// ---- POUs/FBs/FanucKardex/DUTs/ST_Kardex_Robot_Control.TcDUT
TYPE ST_Kardex_Robot_Control :
STRUCT
(*-----=== Byte 01 ===-----*)
	bImmediateStop			:BIT;				// 01.1	Immediate stop
	bHold					:BIT;				// 01.2	Temporary stop
	bSafeSpeed				:BIT;				// 01.3	Safe speed
	bCycleStop				:BIT;				// 01.4	Cycle stop
	bReset					:BIT;				// 01.5	External reset
	bStart					:BIT;				// 01.6	Start
	bHome					:BIT;				// 01.7	Return to home position
	bEnable					:BIT;				// 01.8	Operation enable

(*-----=== Byte 02 ===-----*)
//	nProgNumberSelection	:BYTE;
	bPNS1					:BIT;				// 02.1	Program  number selection
	bPNS2					:BIT;				// 02.2	Program  number selection
	bPNS3					:BIT;				// 02.3	Program  number selection
	bPNS4					:BIT;				// 02.4	Program  number selection
	bPNS5					:BIT;				// 02.5	Program  number selection
	bPNS6					:BIT;				// 02.6	Program  number selection
	bPNS7					:BIT;				// 02.7	Program  number selection
	bPNS8					:BIT;				// 02.8	Program  number selection

(*-----=== Byte 03 ===-----*)
	bPnsStrobe				:BIT;				// 03.1	PNS strobe
	bProdStart				:BIT;				// 03.2	Start of automatic operation
	bZoneEnable				:BIT;				// 03.3	Ez mindig jön kivéve ha vész van
	bServiceEnd				:BIT;				// 03.4	Szervíz üzemmód vége
	{attribute 'hide'}
	_reserved_03_05			:BIT;
	{attribute 'hide'}
	_reserved_03_06			:BIT;
	{attribute 'hide'}
	_reserved_03_07			:BIT;		
	{attribute 'hide'}
	_reserved_03_08			:BIT;		
	
(*-----=== Byte 04 ===-----*)
	{attribute 'hide'}
	_reserved_04			:BYTE;				

(*-----=== Byte 05 ===-----*)
	bKardex_Reset			:BIT;				// 05.1	Robot kardex-be mehet RESET
	bHolder_Reset			:BIT;				// 05.2	Robot Mir-1-be mehet RESET
	bMir_Reset				:BIT;				// 05.3	Robot Mir-2-be mehet RESET
	bPuffer_Reset			:BIT;				// 05.4	Robot pufferbe mehet RESET
	bStrip_1_Reset			:BIT;				// 05.5	Robot szalag-1-be mehet RESET
	bStrip_2_Reset			:BIT;				// 05.6	Robot szalag-2-be mehet RESET
	bStrip_3_Reset			:BIT;				// 05.7	Robot szalag-3-be mehet RESET	
	{attribute 'hide'}
	_reserved_05_08			:BIT;
	
(*-----=== Byte 06 ===-----*)
	{attribute 'hide'}
	_reserved_06			:BYTE;				
	
(*-----=== Byte 07 ===-----*)
	bNotCorrectPrg_Reset			:BIT;				// 07.1	Nem megfelelő mozgási program RESET
	bNotProductOnRobot_Reset		:BIT;				// 07.2	Mozgási program nem hajtható végre, mert a robotnál nincs termék RESET
	bProductOnRobot_Reset			:BIT;				// 07.3	Mozgási program nem hajtható végre, mert a robotnál termék van RESET
	bGripperOpenError_Reset			:BIT;				// 07.4	Megfogó nyitási hiba RESET
	bGripperCloseError_Reset		:BIT;				// 07.5	Megfogó zárási hiba RESET
	bPartPresentError_Reset			:BIT;				// 07.6 Paletta jelenlét hiba RESET
	bNotCorrectKardexFloor_Reset	:BIT;				// 07.7 Nem megfelelő kardex polc RESET
	bNotCorrectKardexJig_Reset		:BIT;				// 07.8 Nem megfelelő kardex üllék RESET

(*-----=== Byte 08 ===-----*)
	bNotCorrectMir_Reset		:BIT;				// 08.1	Nem megfelelő MIR üllék RESET
	bNotCorrectPuffer_Reset		:BIT;				// 08.2 Nem megfelelő puffer üllék RESET
	{attribute 'hide'}
	_reserved_08_03				:BIT;
	{attribute 'hide'}
	_reserved_08_04				:BIT;
	{attribute 'hide'}
	_reserved_08_05				:BIT;
	{attribute 'hide'}
	_reserved_08_06				:BIT;
	{attribute 'hide'}
	_reserved_08_07				:BIT;
	{attribute 'hide'}
	_reserved_08_08				:BIT;

(*-----=== Byte 09-12 ===-----*)
	{attribute 'hide'}
	_reserved_09_12			:ARRAY [9..12] OF BYTE;

(*-----=== Byte 13 ===-----*)
	bPlcOverride			:BYTE;				// 13. PLC által vezérelt sebesség, 10-100 %
	
(*-----=== Byte 14 ===-----*)
	nProgramNumber			:BYTE;				// 14. Mozgatási műveletek kiválasztása.
	
(*-----=== Byte 15 ===-----*)
	nMode					:BYTE;				// 15. PLC által meghatározott robot üzemmód, 1-2
	
(*-----=== Byte 16 ===-----*)
	nKardexFloor			:BYTE;				// 16. Kardex polc szám (1-50)

(*-----=== Byte 17 ===-----*)
	nKardexJig				:BYTE;				// 17. Kardex paletta szám (1-30)
	
(*-----=== Byte 18 ===-----*)
	nMir_1_Jig				:BYTE;				// 18. Mir-1 paletta szám (1-4)
		
(*-----=== Byte 19 ===-----*)
	nMir_2_Jig				:BYTE;				// 19. Mir-2 paletta szám (1-4)
		
(*-----=== Byte 20 ===-----*)
	nPuffer					:BYTE;				// 20. Puffer tároló paletta szám (1-15)
	
(*-----=== Byte 21-64 ===-----*)
	{attribute 'hide'}
	_reserved_21_64			:ARRAY [21..64] OF BYTE;				
END_STRUCT
END_TYPE

// ---- POUs/FBs/FanucKardex/DUTs/ST_Kardex_Robot_Status.TcDUT
TYPE ST_Kardex_Robot_Status :
STRUCT
(*-----=== Byte 01 ===-----*)
	bCommandEnable			:BIT;				// 01.1	During automatic operation
	bSystemReady			:BIT;				// 01.2	Preparation completed
	bProgRun				:BIT;				// 01.3	Program running
	bPaused					:BIT;				// 01.4	Program being interrupted
	bHeld					:BIT;				// 01.5	During temporary stop
	bFault					:BIT;				// 01.6	Alarm
	bHomePos				:BIT;				// 01.7	Home position
	bPendant				:BIT;				// 01.8	Teach pendant enabled

(*-----=== Byte 02 ===-----*)
	bBatteryVoltageDrop		:BIT;				// 02.1	Battery voltage drop
	bBusy					:BIT;				// 02.1	During operation
	bAckSNO1				:BIT;				// 02.1	Selected program number
	bAckSNO2				:BIT;				// 02.2	Selected program number
	bAckSNO3				:BIT;				// 02.3	Selected program number
	bAckSNO4				:BIT;				// 02.4	Selected program number
	bAckSNO5				:BIT;				// 02.5	Selected program number
	bAckSNO6				:BIT;				// 02.6	Selected program number

(*-----=== Byte 03 ===-----*)
	bAckSNO7				:BIT;				// 03.1	Selected program number
	bAckSNO8				:BIT;				// 03.2	Selected program number
	bSnAck					:BIT;				// 03.3	Response signal to PNS
	{attribute 'hide'}
	_reserved_03_04			:BIT;
	bProgramEnd				:BIT;				// 03.5	Robot aktuális programot befejezte
	bProgramRun				:BIT;				// 03.6	Robot aktuális program futásban.
	bAlarm					:BIT;				// 03.7	Robot kűldi amikor hiba van
	bServiceRun				:BIT;				// 03.8 Szerviz pozícióban a robot, szelep vezérlés mehet.
	
(*-----=== Byte 04 ===-----*)
	bGRP_1_2_Open			:BIT;				// 04.1 Megfogó 1&2 nyitva
	bGRP_1_2_Closed			:BIT;				// 04.2 Megfogó 1&2 zárva
	bGRP_3_4_Open			:BIT;				// 04.3 Megfogó 3&4 nyitva
	bGRP_3_4_Closed			:BIT;				// 04.4 Megfogó 3&4 zárva
	bPartPresent			:BIT;				// 04.5 Paletta figyelő/bemérő szenzor
	{attribute 'hide'}
	_reserved_04_06			:BIT;				
	{attribute 'hide'}
	_reserved_04_07			:BIT;
	{attribute 'hide'}
	_reserved_04_08			:BIT;
	
(*-----=== Byte 05 ===-----*)
	bKardex_Set				:BIT;				// 05.1	Robot kardex-be menne SET
	bHolder_Set				:BIT;				// 05.2	Robot Mir-1-be menne SET
	bMir_Set				:BIT;				// 05.3	Robot Mir-2-be menne SET
	bPuffer_Set				:BIT;				// 05.4	Robot pufferbe menne SET
	bStrip_1_Set			:BIT;				// 05.5	Robot szalag-1-be menne SET
	bStrip_2_Set			:BIT;				// 05.6	Robot szalag-2-be menne SET
	bStrip_3_Set			:BIT;				// 05.7	Robot szalag-3-be menne SET	
	{attribute 'hide'}
	_reserved_05_08			:BIT;
	
(*-----=== Byte 06 ===-----*)
	{attribute 'hide'}
	_reserved_06			:BYTE;				
	
(*-----=== Byte 07 ===-----*)
	bNotCorrectPrg					:BIT;		// 07.1	Nem megfelelő mozgási program SET
	bNotProductOnRobot				:BIT;		// 07.2	Mozgási program nem hajtható végre, mert a robotnál nincs termék SET
	bProductOnRobot					:BIT;		// 07.3	Mozgási program nem hajtható végre, mert a robotnál termék van SET
	bGripperOpenError				:BIT;		// 07.4	Megfogó nyitási hiba SET
	bGripperCloseError				:BIT;		// 07.5 Megfogó zárási hiba SET
	bPartPresentError				:BIT;		// 07.6 Paletta jelenlét hiba SET
	bNotCorrectKardexFloor			:BIT;		// 07.7 Nem megfelelő kardex polc SET
	bNotCorrectKardexJig			:BIT;		// 07.8 Nem megfelelő kardex üllék SET

(*-----=== Byte 08 ===-----*)
	bNotCorrectMir				:BIT;			// 08.1	Nem megfelelő MIR üllék SET
	bNotCorrectPuffer			:BIT;			// 08.2 Nem megfelelő puffer üllék SET
	{attribute 'hide'}
	_reserved_08_03				:BIT;
	{attribute 'hide'}
	_reserved_08_04				:BIT;
	{attribute 'hide'}
	_reserved_08_05				:BIT;
	{attribute 'hide'}
	_reserved_08_06				:BIT;
	{attribute 'hide'}
	_reserved_08_07				:BIT;
	{attribute 'hide'}
	_reserved_08_08				:BIT;
	
(*-----=== Byte 09 ===-----*)
	bZone_1_Kardex			:BIT;				// 09.1	Robot bent a területen. - Kardex
	bZone_2_Holder			:BIT;				// 09.2	Robot bent a területen. - Mir1
	bZone_3_Mir1			:BIT;				// 09.3	Robot bent a területen. - Mir2
	bZone_4_Puffer			:BIT;				// 09.4	Robot bent a területen. - Puffer
	bZone_5_Strip			:BIT;				// 09.5	Robot bent a területen. - Szalag
	bZone_6_Trans			:BIT;				// 09.6	Robot bent a területen. - Átmozgási terület
	{attribute 'hide'}
	_reserved_09_07			:BIT;		
	{attribute 'hide'}
	_reserved_09_08			:BIT;	
	
(*-----=== Byte 09 ===-----*)
	bRobotInStrip_1			:BIT;				// 10.1	Robot bent a szalag-1-ben.
	bRobotInStrip_2			:BIT;				// 10.2	Robot bent a szalag-2-ben.
	bRobotInStrip_3			:BIT;				// 10.3	Robot bent a szalag-3-ban.
	{attribute 'hide'}
	_reserved_10_04			:BIT;	
	{attribute 'hide'}
	_reserved_10_05			:BIT;		
	{attribute 'hide'}
	_reserved_10_06			:BIT;	
	{attribute 'hide'}
	_reserved_10_07			:BIT;		
	{attribute 'hide'}
	_reserved_10_08			:BIT;	

(*-----=== Byte 11 - 12 ===-----*)
	{attribute 'hide'}
	_reserved_10_12			:ARRAY[11..12] OF BYTE;				
	
(*-----=== Byte 13 ===-----*)
	nProgramNumber			:BYTE;				// 13. Aktuális program szám Robotban,
	
(*-----=== Byte 14 ===-----*)
	nPointNumber			:BYTE;				// 14. Aktuális pont szám
	
(*-----=== Byte 15 ===-----*)
	bKeyAuto				:BIT;				// 15.1	Robot automata-remote üzemmódban
	bKeyManualT1			:BIT;				// 15.2	Robot kézi üzemmódban - 250 mm/sec max sebesség
	bKeyManualT2			:BIT;				// 15.3	Robot kézi üzemmódban - 100 % sebesség
	bSimInput				:BIT;				// 15.4	Szimulálva (force-olva) Input
	bSimOutput				:BIT;				// 15.5	Szimulálva (force-olva) Output
	{attribute 'hide'}
	_reserved_15_06			:BIT;
	{attribute 'hide'}
	_reserved_15_07			:BIT;		
	{attribute 'hide'}
	_reserved_15_08			:BIT;	
	
(*-----=== Byte 16 ===-----*)
	bControllerEmyStop		:BIT;				// 16.1	Robot kontroller vészgomb
	bTeachPendantEmyStop	:BIT;				// 16.2	Teach Pendant vészgomb
	bDeadman				:BIT;				// 16.3	TP engedélyező gomb
	bFence					:BIT;				// 16.4	Fence
	bRot					:BIT;				// 16.5	Robot olyan területre akar mozogni ahova mechanikusan nem ér el
	bHbk					:BIT;				// 16.6	Robot felütközött, védelem
	bEmyStopExternal		:BIT;				// 16.7	Külső vészgomb (gépi)
	bNoPneumatics			:BIT;				// 16.8	A karon lévő pneumatika nem érzékel levegőt
	
(*-----=== Byte 17 ===-----*)
	bBeltBreak				:BIT;				// 17.1	Robot kontroller vészgomb
	bFalm					:BIT;				// 17.2	Ventilátor hiba
	bServoOff				:BIT;				// 17.3	Kivűlről tiltott SERVO engedélyezés
	bIMSTP					:BIT;				// 17.4	Engedélyező jel vissza adása
	bBEKHLD					:BIT;				// 17.5	
	bUSRALM					:BIT;				// 17.6	
	bSRVDSCNCT				:BIT;				// 17.7	
	bNTED					:BIT;				// 17.8			
	
(*-----=== Byte 18 - 64 ===-----*)
	{attribute 'hide'}
	_reserved_18_64			:ARRAY[18..64] OF BYTE;		
END_STRUCT
END_TYPE

// ---- POUs/FBs/FanucKardex/DUTs/U_Kardex_Fanuc_Input.TcDUT
TYPE U_Kardex_Fanuc_Input :
UNION
	aStdIn		AT %I*		:ARRAY [1..32] OF UINT;
	Status					:ST_Kardex_Robot_Status;	
END_UNION
END_TYPE

// ---- POUs/FBs/FanucKardex/DUTs/U_Kardex_Fanuc_Output.TcDUT
TYPE U_Kardex_Fanuc_Output :
UNION
	aStdOut		AT %Q*		:ARRAY [1..32] OF UINT;
	Control					:ST_Kardex_Robot_Control;	
END_UNION
END_TYPE

// ---- POUs/FBs/Fanuc/DUTs/E_Robot_Command.TcDUT
{attribute 'qualified_only'}
{attribute 'strict'}
TYPE E_Robot_Command :
(
	NoCommand 				:= 0,
	Home					:= 1,
	Wait					:= 2,
	Service					:= 3,
	Pick_Up_Vise			:= 4,
	Put_Down_Vise			:= 5,
	Pick_Up_Cnc 			:= 6,
	Put_Down_Cnc 			:= 7,
	Move_To_Clean			:= 8
);
END_TYPE

// ---- POUs/FBs/Fanuc/DUTs/E_Robot_Programs.TcTLEO
{attribute 'strict'}
{attribute 'to_string'}
TYPE E_Robot_Programs :
(
	NoCommand			:= 0,
	Home				:= 1,
	Park				:= 2,
	Service				:= 3,
	VisePickUp_1_7 		:= 11,
	VisePutDown_1_7 	:= 12,
	VisePickUp_8_14		:= 13,
	VisePutDown_8_14	:= 14,
	VisePutDownToCnc_4 	:= 15,
	VisePickUpFromCnc_4	:= 16,
	VisePutDownToCnc_5	:= 17,
	VisePickUpFromCnc_5	:= 18
);
END_TYPE

// ---- POUs/FBs/Fanuc/DUTs/ST_Robot_Status.TcDUT
TYPE ST_Robot_Status :
STRUCT
(*-----=== Byte 01 ===-----*)
	bCommandEnable			:BIT;				// 01.1	During automatic operation
	bSystemReady			:BIT;				// 01.2	Preparation completed
	bProgRun				:BIT;				// 01.3	Program running
	bPaused					:BIT;				// 01.4	Program being interrupted
	bHeld					:BIT;				// 01.5	During temporary stop
	bFault					:BIT;				// 01.6	Alarm
	bHomePos				:BIT;				// 01.7	Home position
	bPendant				:BIT;				// 01.8	Teach pendant enabled

(*-----=== Byte 02 ===-----*)
	bBatteryVoltageDrop		:BIT;				// 02.1	Battery voltage drop
	bBusy					:BIT;				// 02.2	During operation
	bAckSNO1				:BIT;				// 02.3	Selected program number
	bAckSNO2				:BIT;				// 02.4	Selected program number
	bAckSNO3				:BIT;				// 02.5	Selected program number
	bAckSNO4				:BIT;				// 02.6	Selected program number
	bAckSNO5				:BIT;				// 02.7	Selected program number
	bAckSNO6				:BIT;				// 02.8	Selected program number

(*-----=== Byte 03 ===-----*)
	bAckSNO7				:BIT;				// 03.1	Selected program number
	bAckSNO8				:BIT;				// 03.2	Selected program number
	bSnAck					:BIT;				// 03.3	Response signal to PNS
	{attribute 'hide'}
	_reserved_03_04			:BIT;
	bProgramEnd				:BIT;				// 03.5	Robot aktuális programot befejezte
	bProgramRun				:BIT;				// 03.6	Robot aktuális program futásban.
	bAlarm					:BIT;				// 03.7	Robot kűldi amikor hiba van
	bServiceRun				:BIT;				// 03.8 Szerviz pozícióban a robot, szelep vezérlés mehet.
	
(*-----=== Byte 04 ===-----*)
	bGripperOpen			:BIT;				// 04.1	Robot IO, gripper nyitva
	bGripperClose			:BIT;				// 04.2	Robot IO, gripper zárva
	bVisePresent			:BIT;				// 04.3	Robot IO, satu a megfogóban
	{attribute 'hide'}
	_reserved_04_04			:BIT;
	{attribute 'hide'}
	_reserved_04_05			:BIT;
	{attribute 'hide'}
	_reserved_04_06			:BIT;
	{attribute 'hide'}
	_reserved_04_07			:BIT;		
	{attribute 'hide'}
	_reserved_04_08			:BIT;

(*-----=== Byte 05 ===-----*)
	bVise_1_7_Set			:BIT;				// 05.1	Robot satú 1-7-be menne SET
	bVise_8_14_Set			:BIT;				// 05.2	Robot satú 8-14-be menne SET
	bCNC_4_Set				:BIT;				// 05.3	Robot CNC-4-be menne SET
	bCNC_5_Set				:BIT;				// 05.4	Robot CNC-5-be menne SET
	{attribute 'hide'}
	_reserved_05_05			:BIT;
	{attribute 'hide'}
	_reserved_05_06			:BIT;
	{attribute 'hide'}
	_reserved_05_07			:BIT;		
	{attribute 'hide'}
	_reserved_05_08			:BIT;
	
(*-----=== Byte 06 ===-----*)
	{attribute 'hide'}
	_reserved_06			:BYTE;				
	
(*-----=== Byte 07 ===-----*)
	bNotCorrectPrg			:BIT;				// 07.1	Nem megfelelő mozgási program SET
	bNotProductOnRobot		:BIT;				// 07.2	Mozgási program nem hajtható végre, mert a robotnál nincs termék SET
	bProductOnRobot			:BIT;				// 07.3	Mozgási program nem hajtható végre, mert a robotnál termék van SET
	bGripperOpenError		:BIT;				// 07.4	Megfogó nyitási hiba SET
	bGripperCloseError		:BIT;				// 07.5 Megfogó zárási hiba SET
	bNotCorrectViseNumber	:BIT;				// 07.6 Nem megfelelő satú sorszám SET
	{attribute 'hide'}
	_reserved_07_07			:BIT;		
	{attribute 'hide'}
	_reserved_07_08			:BIT;	

(*-----=== Byte 08 ===-----*)
	{attribute 'hide'}
	_reserved_08			:BYTE;
	
(*-----=== Byte 09 ===-----*)
	bZone_1_Vise_1_7		:BIT;				// 09.1	Robot bent a területen.
	bZone_2_Vise_8_14		:BIT;				// 09.2	Robot bent a területen.
	bZone_3_Trans			:BIT;				// 09.3	Robot bent a területen.
	bZone_4_CNC_4			:BIT;				// 09.4	Robot bent a területen.
	bZone_5_CNC_5			:BIT;				// 09.5	Robot bent a területen.
	{attribute 'hide'}
	_reserved_09_06			:BIT;
	{attribute 'hide'}
	_reserved_09_07			:BIT;		
	{attribute 'hide'}
	_reserved_09_08			:BIT;	

(*-----=== Byte 10 ===-----*)
	{attribute 'hide'}
	_reserved_10			:BYTE;

(*-----=== Byte 11 ===-----*)
	{attribute 'hide'}
	_reserved_11			:BYTE;

(*-----=== Byte 12 ===-----*)
	{attribute 'hide'}
	_reserved_12			:BYTE;
	
(*-----=== Byte 13 ===-----*)
	nProgramNumber			:BYTE;				// 13. Aktuális program szám Robotban,
	
(*-----=== Byte 14 ===-----*)
	nPointNumber			:BYTE;				// 14. Aktuális pont szám
	
(*-----=== Byte 15 ===-----*)
	bKeyAuto				:BIT;				// 15.1	Robot automata-remote üzemmódban
	bKeyManualT1			:BIT;				// 15.2	Robot kézi üzemmódban - 250 mm/sec max sebesség
	bKeyManualT2			:BIT;				// 15.3	Robot kézi üzemmódban - 100 % sebesség
	bSimInput				:BIT;				// 15.4	Szimulálva (force-olva) Input
	bSimOutput				:BIT;				// 15.5	Szimulálva (force-olva) Output
	{attribute 'hide'}
	_reserved_15_06			:BIT;
	{attribute 'hide'}
	_reserved_15_07			:BIT;		
	{attribute 'hide'}
	_reserved_15_08			:BIT;	
	
(*-----=== Byte 16 ===-----*)
	bControllerEmyStop		:BIT;				// 16.1	Robot kontroller vészgomb
	bTeachPendantEmyStop	:BIT;				// 16.2	Teach Pendant vészgomb
	bDeadman				:BIT;				// 16.3	TP engedélyező gomb
	bFence					:BIT;				// 16.4	Fence
	bRot					:BIT;				// 16.5	Robot olyan területre akar mozogni ahova mechanikusan nem ér el
	bHbk					:BIT;				// 16.6	Robot felütközött, védelem
	bEmyStopExternal		:BIT;				// 16.7	Külső vészgomb (gépi)
	bNoPneumatics			:BIT;				// 16.8	A karon lévő pneumatika nem érzékel levegőt
	
(*-----=== Byte 17 ===-----*)
	bBeltBreak				:BIT;				// 17.1	Robot kontroller vészgomb
	bFalm					:BIT;				// 17.2	Ventilátor hiba
	bServoOff				:BIT;				// 17.3	Kivűlről tiltott SERVO engedélyezés
	bIMSTP					:BIT;				// 17.4	Engedélyező jel vissza adása
	bBEKHLD					:BIT;				// 17.5	
	bUSRALM					:BIT;				// 17.6	
	bSRVDSCNCT				:BIT;				// 17.7	
	bNTED					:BIT;				// 17.8			
	
(*-----=== Byte 17 - 64 ===-----*)
	{attribute 'hide'}
	_reserved_17_64			:ARRAY[17..64] OF BYTE;		
END_STRUCT
END_TYPE

// ---- POUs/FBs/Fanuc/DUTs/U_Fanuc_Input.TcDUT
TYPE U_Fanuc_Input :
UNION
	aStdIn		AT %I*		:ARRAY [1..32] OF UINT;
	Status					:ST_Robot_Status;	
END_UNION
END_TYPE

// ---- POUs/FBs/Fanuc/DUTs/U_Fanuc_Output.TcDUT
TYPE U_Fanuc_Output :
UNION
	aStdOut		AT %Q*		:ARRAY [1..32] OF UINT;
	Control					:ST_Robot_Control;	
END_UNION
END_TYPE

// ---- POUs/FBs/ID200/DUTs/E_CarrierType.TcTLEO
{attribute 'qualified_only'}
{attribute 'strict'}
TYPE E_CarrierType :
(
	EM4102		:= 16#3032,
	EM4550		:= 16#3033,
	Nova		:= 16#3130,
	Q5			:= 16#3131,
	T5557		:= 16#3134,
	MDT_28		:= 16#3135,
	ISO15693	:= 16#3230,
	MDT_112		:= 16#3231,
	TiHF_I		:= 16#3232,
	SRF55V02P	:= 16#3233,
	SRF55V10P	:= 16#3234,
	MDT_2K_H	:= 16#3333,
	SLI_S		:= 16#3335,
	Depending	:= 16#3939
)WORD := MDT_28;
END_TYPE
//  EM4102 = '16#3032'
//  EM4550 = '16#3033'
//  Nova = '16#3130'
//  Q5 = '16#3131'
//  T5557 = '16#3134'
//  MDT_28 = '16#3135'
//  ISO15693 = '16#3230'
//  MDT_112 = '16#3231'
//  TiHF_I = '16#3232'
//  SRF55V02P = '16#3233'
//  SRF55V10P = '16#3234'
//  MDT_2K_H = '16#3333'
//  SLI_S = '16#3335'
//  Depending = '16#3939'

// ---- POUs/FBs/ID200/DUTs/E_Command.TcTLEO
{attribute 'qualified_only'}
{attribute 'strict'}
TYPE E_Command :
(
	Quit := 16#02,
	ChangeTag := 16#04,
	Reset := 16#16,
	SetMultiplexedMode := 16#9B,
	SetTriggerMode := 16#9C,
	SingleReadFixCode := 16#01,
	EnchancedReadFixCode := 16#1D,
	SingleReadWords := 16#10,
	EnchancedReadWords := 16#19,
	SingleWriteWords := 16#40,
	SingleWriteFixCode := 16#1F
)BYTE := Quit;
END_TYPE
//  Quit = '16#02'
//  ChangeTag = '16#04'
//  Reset = '16#16'
//  SetMultiplexedMode = '16#9B'
//  SetTriggerMode = '16#9C'
//  SingleReadFixCode = '16#01'
//  EnchancedReadFixCode = '16#1D'
//  SingleReadWords = '16#10'
//  EnchancedReadWords = '16#19'
//  SingleWriteWords = '16#40'
//  SingleWriteFixCode = '16#1F'

// ---- POUs/FBs/ID200/DUTs/E_TagStatus.TcTLEO
{attribute 'qualified_only'}
{attribute 'strict'}
TYPE E_TagStatus :
(
	NotPresent	:= 0,
	FixCode		:= 1,
	UserCode	:= 2
)BYTE := NotPresent;
END_TYPE

// ---- POUs/FBs/ID200/DUTs/RawToUlint.TcDUT
TYPE RawToUlint :
UNION
	Number		: ULINT;
	Raw			: ARRAY [0..7] OF BYTE;
END_UNION
END_TYPE

// ---- POUs/FBs/ID200/DUTs/ST_Active_RFIDs.TcDUT
TYPE ST_Active_RFIDs :
STRUCT
	RFID			: INT;
	CH				: BYTE;
END_STRUCT
END_TYPE

// ---- POUs/FBs/ID200/DUTs/ST_Tag_Data.TcDUT
TYPE ST_Tag_Data :
STRUCT
	Status			: E_TagStatus;
	RawData			: ARRAY [0..7] OF BYTE;
	Code			: ULINT;
END_STRUCT
END_TYPE

// ---- POUs/FBs/ID200/DUTs/WordToBytes.TcDUT
TYPE WordToBytes :
UNION
	word_in			: WORD;
	bytes			: ARRAY [0..1] OF BYTE;
END_UNION
END_TYPE

// ---- POUs/FBs/MPS/DUTs/U_to_int.TcDUT
TYPE U_to_int :
UNION
	arrRaw			: ARRAY [0..1] OF BITARR8;
	nData			: INT;
END_UNION
END_TYPE

// ---- POUs/FBs/MySQL/NextVise/DUTs/ST_ParaVal_GetNextVise.TcDUT
TYPE ST_ParaVal_GetNextVise :
STRUCT
	Target			: BYTE;
	ViseNumber		: BYTE;
END_STRUCT
END_TYPE

// ---- POUs/FBs/MySQL/SetViseState/DUTs/ST_ParaVal_SetViseStae.TcDUT
TYPE ST_ParaVal_SetViseStae :
STRUCT
	Target			: BYTE;
	ViseNumber		: BYTE;
END_STRUCT
END_TYPE

// ---- POUs/FBs/MySQL/UpdateVise/DUTs/ST_ParaVal_UpdateVise.TcDUT
TYPE ST_ParaVal_UpdateVise :
STRUCT
	ViseNumber			: SINT;
	SerialNumber		: STRING(255);
	DutIdentifier		: LINT;
	CamIdentifier		: LINT;
	CncNumber			: SINT;
END_STRUCT
END_TYPE

// ---- POUs/FBs/ServoVise/DUTs/E_ServoVise_Command.TcTLEO
{attribute 'qualified_only'}
{attribute 'strict'}
TYPE E_ServoVise_Command :
(
	NoCommand,
	Attach,
	MoveToPos,
	Release,
	Fix
);
END_TYPE

// ---- POUs/FBs/ServoVise/DUTs/E_ViseJawState.TcTLEO
{attribute 'qualified_only'}
{attribute 'strict'}
TYPE E_ViseJawState :
(
	P1_0_120,
	P2_80_210
);
END_TYPE

// ---- POUs/Temp/Fanuc/E_Fanuc_Program.TcDUT
{attribute 'strict'}
TYPE E_Fanuc_Program :
(
	NoCommand := 0,					// Üres utasítás
	Home := 1,						// Alaphelyzet felvétel
	Service1 := 2,					// Szerviz pozíció 1
	Service2 := 3,					// Szerviz pozíció 2
	Service3 := 4,					// Szerviz pozíció 3
	PickUpFeeder1 := 5,				// Alkatrész felvétel Feeder1-ből
	PickUpFeeder2 := 6,				// Alkatrész felvétel Feeder2-ből
	PickUpFeeder3 := 7,				// Alkatrész felvétel Feeder3-ból
	PickUpFeeder4 := 8,				// Alkatrész felvétel Feeder4-ből
	PutDownPositioner1 := 9,		// Alkatrész lerakás 1. tájolóba
	PickUpPositioner1 := 10,		// Alkatrész felvéte 1. tájolóból
	PutDownPositioner2 := 11,		// Alkatrész lerakás 2. tájolóba
	PickUpPositioner2 := 12,		// Alkatrész felvétel 2. tájolóból
	PressCamCoord := 13,			// Alkatrész préselés küldött pozícióra
	PressFixCoord1 := 14,			// Alkatrész préselés Fix pozícióra 1
	PressFixCoord2 := 15,			// Alkatrész préselés Fix pozícióra 2
	PressFixCoord3 := 16,			// Alkatrész préselés Fix pozícióra 3
	PressFixCoord4 := 17,			// Alkatrész préselés Fix pozícióra 4
	TempPos := 18,					// Várakozó pozíció
	OriginCalibA := 19,				// Robot présfej mozgatása kalibráló ülék fölé (Kézi 0 pont állítás)
	OriginCalibB := 20,				// Aktuális pozícióra robot offset beállítása
	CalibPositioner1 := 21,			// Tájoló 1-ből alkatrész kiszedés kalibráló lapra lerakás koordináták elküldése
	CalibPositioner2 := 22,			// Tájoló 1-ből alkatrész kiszedés kalibráló lapra lerakás koordináták elküldése
	CalibPickUpStoreS1 := 23,		// Kicsi 1. kalibráló darab felvétele a tárolóból
	CalibPickUpStoreS2 := 24,		// Kicsi 2. kalibráló darab felvétele a tárolóból
	CalibPickUpStoreS3 := 25,		// Kicsi 3. kalibráló darab felvétele a tárolóból
	CalibPickUpStoreS4 := 26,		// Kicsi 4. kalibráló darab felvétele a tárolóból
	CalibPutDownStoreS1 := 27,		// Kicsi 1. kalibráló darab lerakása a tárolóba
	CalibPutDownStoreS2 := 28,		// Kicsi 2. kalibráló darab lerakása a tárolóba
	CalibPutDownStoreS3 := 29,		// Kicsi 3. kalibráló darab lerakása a tárolóba
	CalibPutDownStoreS4 := 30,		// Kicsi 4. kalibráló darab lerakása a tárolóba
	CalibPickUpStoreL1 := 31,		// Nagy 1. kalibráló darab felvétele a tárolóból
	CalibPickUpStoreL2 := 32,		// Nagy 2. kalibráló darab felvétele a tárolóból
	CalibPickUpStoreL3 := 33,		// Nagy 3. kalibráló darab felvétele a tárolóból
	CalibPickUpStoreL4 := 34,		// Nagy 4. kalibráló darab felvétele a tárolóból
	CalibPutDownStoreL1 := 35,		// Nagy 1. kalibráló darab lerakása a tárolóba
	CalibPutDownStoreL2 := 36,		// Nagy 2. kalibráló darab lerakása a tárolóba
	CalibPutDownStoreL3 := 37,		// Nagy 3. kalibráló darab lerakása a tárolóba
	CalibPutDownStoreL4 := 38,		// Nagy 4. kalibráló darab lerakása a tárolóba
	CalibPutDownUpper1 := 39,		// Kalibráló darab lerakás felső lap 1. pozícióba
	CalibPutDownUpper2 := 40,		// Kalibráló darab lerakás felső lap 2. pozícióba
	CalibPutDownUpper3 := 41,		// Kalibráló darab lerakás felső lap 3. pozícióba
	CalibPutDownUpper4 := 42,		// Kalibráló darab lerakás felső lap 4. pozícióba
	CalibPickUpUpper1 := 43,		// Kalibráló darab felvétel felső lap 1. pozícióból
	CalibPickUpUpper2 := 44,		// Kalibráló darab felvétel felső lap 2. pozícióból
	CalibPickUpUpper3 := 45,		// Kalibráló darab felvétel felső lap 3. pozícióból
	CalibPickUpUpper4 := 46,		// Kalibráló darab felvétel felső lap 4. pozícióból
	CalibPutDownLower1 := 47,		// Kalibráló darab lerakás alsó lap 1. pozícióba
	CalibPutDownLower2 := 48,		// Kalibráló darab lerakás alsó lap 2. pozícióba
	CalibPutDownLower3 := 49,		// Kalibráló darab lerakás alsó lap 3. pozícióba
	CalibPutDownLower4 := 50,		// Kalibráló darab lerakás alsó lap 4. pozícióba
	CalibPickUpLower1 := 51,		// Kalibráló darab felvétel alsó lap 1. pozícióból
	CalibPickUpLower2 := 52,		// Kalibráló darab felvétel alsó lap 2. pozícióból
	CalibPickUpLower3 := 53,		// Kalibráló darab felvétel alsó lap 3. pozícióból
	CalibPickUpLower4 := 54,		// Kalibráló darab felvétel alsó lap 4. pozícióból
	CalibPickUpPositioner1 := 55,	// Kalibráló darab felvétel 1. tájolóból
	CalibPickUpPositioner2 := 56	// Kalibráló darab felvétel 2. tájolóból
) := NoCommand;
END_TYPE

// ---- POUs/Temp/Fanuc/ST_FanucReq.TcDUT
TYPE ST_FanucReq :
STRUCT
	nProgNr					:Byte;				
	nMovePoint				:BYTE;
	sName					:STRING;
END_STRUCT
END_TYPE

// ---- POUs/Temp/Fanuc/ST_Fanuc_Alarm_In.TcDUT
TYPE ST_Fanuc_Alarm_In :
STRUCT
	(* -----=== Byte 06 ===----- *)
	bAlarm1						:BIT;			//	Program hívási hiba: A robot nem fog terméket
	bAlarm2						:BIT;			//	Program hívási hiba: A robot terméket fog
	bAlarm3						:BIT;			//	Program hívási hiba: Nincs ilyen program
	bAlarm4						:BIT;			//	Termék megfogás hiba: Vákuum hiba átrakó
	bAlarm5						:BIT;			//	Termék fogás hiba: Vákuum hiba prés
	bAlarm6						:BIT;			//	Préselés: Folyamat megszakítva, erőmérés hiba
	{attribute 'hide'}
	_reserved_06_7				:BIT;			// Tartalék 06.07	
	{attribute 'hide'}
	_reserved_06_8				:BIT;			// Tartalék 06.08	
END_STRUCT
END_TYPE

// ---- POUs/Temp/Fanuc/ST_Fanuc_Alarm_Out.TcDUT
TYPE ST_Fanuc_Alarm_Out :
STRUCT
	(* -----=== Byte 06 ===----- *)
	bAlarm1						:BIT;			//	Program hívási hiba: A robot nem fog terméket
	bAlarm2						:BIT;			//	Program hívási hiba: A robot terméket fog
	bAlarm3						:BIT;			//	Program hívási hiba: Nincs ilyen program
	bAlarm4						:BIT;			//	Termék megfogás hiba: Vákuum hiba átrakó
	bAlarm5						:BIT;			//	Termék fogás hiba: Vákuum hiba prés
	bAlarm6						:BIT;			//	Préselés: Folyamat megszakítva, erőmérés hiba
	{attribute 'hide'}
	_reserved_06_7				:BIT;			// Tartalék 06.07	
	{attribute 'hide'}
	_reserved_06_8				:BIT;			// Tartalék 06.08	
END_STRUCT
END_TYPE

// ---- POUs/Temp/Fanuc/ST_Fanuc_Area_In.TcDUT
TYPE ST_Fanuc_Area_In :
STRUCT
	(* -----=== Byte 03 ===----- *)
	bFeeder						:BIT;			//	Robot a Fuji adaagolóknál
	bPositioner1				:BIT;			//	Tájoló 1-nél
	bPositioner2				:BIT;			//	Tájoló 2-nél
	bFixtureArea				:BIT;			//	PCB üléknél
	{attribute 'hide'}
	_reserved_03_5				:BIT;			// Tartalék 03.05	
	{attribute 'hide'}
	_reserved_03_6				:BIT;			// Tartalék 03.06	
	{attribute 'hide'}
	_reserved_03_7				:BIT;			// Tartalék 03.07	
	{attribute 'hide'}
	_reserved_03_8				:BIT;			// Tartalék 03.08	
END_STRUCT
END_TYPE

// ---- POUs/Temp/Fanuc/ST_Fanuc_Control_In.TcDUT
TYPE ST_Fanuc_Control_In :
STRUCT
	(* -----=== Byte 01 ===----- *)
	bCmdEnable					:BIT;			//	A robot automata módba van
	bFault						:BIT;			//	A robot hiba
	bBattery					:BIT;			//	A robot elem figyelmeztetés
	bBusy						:BIT;			//	A robot elfoglalt
	bProgEnd					:BIT;			//	Aktuális program kész
	bProgRun					:BIT;			//	Aktuális program fut
	bError						:BIT;			//	Program hiba
	bServiceRun					:BIT;			//	Robot szervíz pozícióban
END_STRUCT
END_TYPE

// ---- POUs/Temp/Fanuc/ST_Fanuc_Control_Out.TcDUT
TYPE ST_Fanuc_Control_Out :
STRUCT
	(* -----=== Byte 01 ===----- *)
	bImStop						:BIT;			//	Immediate stop			Mindig kint van kivéve vészstop (Alacsony aktív)
	bHold						:BIT;			//	Temporary stop			Mindig kint van kivéve vészstop (Alacsony aktív)
	bSafetyfSpeed				:BIT;			//	Safety speed			Mindig kint van kivéve vészstop (Alacsony aktív)
	bCycleStop					:BIT;			//	Cycle stop
	bReset						:BIT;			//	External reset			Robot hibatörlés, nem alarm
	bStart						:BIT;			//	Cycle start
	bEnable						:BIT;			//	Operational enable
	bPsr1						:BIT;			//	Prg 1					Nincs használva
	(* -----=== Byte 02 ===----- *)	
	bPsr2						:BIT;			//	Prg 2					Nincs használva
	bPsr3						:BIT;			//	Prg 3					Nincs használva
	bPsr4						:BIT;			//	Prg 4					Nincs használva
	bPsrStrobe					:BIT;			//	Prg strobe				Nincs használva
	bMoveEnable					:BIT;			//	Move enable				Mindig kint van kivéve vészstop (Alacsony aktív)
	bServiceEnd					:BIT;			//	Sevice end
	{attribute 'hide'}
	_reserved_02_7				:BIT;			// Tartalék 02.07	
	{attribute 'hide'}
	_reserved_02_8				:BIT;			// Tartalék 02.08	
END_STRUCT
END_TYPE

// ---- POUs/Temp/Fanuc/ST_Fanuc_Data_In.TcDUT
TYPE ST_Fanuc_Data_In :
STRUCT
	(* -----=== Byte 07, 08 ===----- *)
	nPositionX					:WORD;			//	Formátuma egész pozítiv szám. A felhasználása szám/100. Pl.: 123,45 > 12345
	(* -----=== Byte 09, 10 ===----- *)
	nPositionY					:WORD;			//	Formátuma egész pozítiv szám. A felhasználása szám/100. Pl.: 123,45 > 12345
	(* -----=== Byte 11, 12 ===----- *)
	nPositionR					:WORD;			//	
END_STRUCT
END_TYPE

// ---- POUs/Temp/Fanuc/ST_Fanuc_Data_Out.TcDUT
TYPE ST_Fanuc_Data_Out :
STRUCT
	(* -----=== Byte 08, 09 ===----- *)
	nPositionX					:WORD;			//	Formátuma egész pozítiv szám. A felhasználása szám/100. Pl.: 123,45 > 12345
	(* -----=== Byte 10, 11 ===----- *)
	nPositionY					:WORD;			//	Formátuma egész pozítiv szám. A felhasználása szám/100. Pl.: 123,45 > 12345
	(* -----=== Byte 12, 13 ===----- *)
	nPositionR					:WORD;			//	
END_STRUCT
END_TYPE

// ---- POUs/Temp/Fanuc/ST_Fanuc_DIO_In.TcDUT
TYPE ST_Fanuc_DIO_In :
STRUCT
	(* -----=== Byte 04 ===----- *)
	bVacuumPressOK				:BIT;			//	Vákuum présfej visszajelzés
	bVacuumMoveOK				:BIT;			//	Vákuum átrakó visszajelzés
	bMoverUp					:BIT;			//	Átrakó henger fent
	bMoverDown					:BIT;			//	Átrakó henger lent
	{attribute 'hide'}
	_reserved_04_5				:BIT;			// Tartalék 04.05	
	{attribute 'hide'}
	_reserved_04_6				:BIT;			// Tartalék 04.06	
	{attribute 'hide'}
	_reserved_04_7				:BIT;			// Tartalék 04.07	
	{attribute 'hide'}
	_reserved_04_8				:BIT;			// Tartalék 04.08	

	(* -----=== Byte 05 ===----- *)
	bVacuumPressOn				:BIT;			//	Présfej vákuum bekapcsolva
	bVacuumMoveOn				:BIT;			//	Átrakó vákuum bekapcsolva
	bMoverUpOn					:BIT;			//	Átrakó henger fel
	bMoverDownOn				:BIT;			//	Átrakó henger le
	{attribute 'hide'}
	_reserved_05_5				:BIT;			// Tartalék 05.05	
	{attribute 'hide'}
	_reserved_05_6				:BIT;			// Tartalék 05.06	
	{attribute 'hide'}
	_reserved_05_7				:BIT;			// Tartalék 05.07	
	{attribute 'hide'}
	_reserved_05_8				:BIT;			// Tartalék 05.08	
END_STRUCT
END_TYPE

// ---- POUs/Temp/Fanuc/ST_Fanuc_Emergency_In.TcDUT
TYPE ST_Fanuc_Emergency_In :
STRUCT
	(* -----=== Byte 15 ===----- *)
	bEMGOP						:BIT;			//	Robot kontroller vészgomb
	bEMGTP						:BIT;			//	Teach Pendant vészgomb
	bDEADMAN					:BIT;			//	TP engedélyező gomb
	bFENCE						:BIT;			//	Fence
	bROT						:BIT;			//	Robot olyan területre akar mozogni ahova mechanikusan nem ér el
	bHBK						:BIT;			//	Robot felütközött, védelem
	bEMGEX						:BIT;			//	Külső vészgomb (gépi)
	bPPABN						:BIT;			//	A karon lévő pneumatika nem érzékel levegőt
	(* -----=== Byte 16 ===----- *)
	bBELTBREAK					:BIT;			//	
	bFALM						:BIT;			//	Ventilátor hiba
	bSVOFF						:BIT;			//	Kivűlről tiltott SERVO engedélyezés
	bIMSTP						:BIT;			//	Engedélyező jel vissza adása
	bBEKHLD						:BIT;				
	bUSRALM						:BIT;				
	bSRVDSCNCT					:BIT;				
	bNTED						:BIT;				
END_STRUCT
END_TYPE

// ---- POUs/Temp/Fanuc/ST_Fanuc_HandShake_In.TcDUT
TYPE ST_Fanuc_HandShake_In :
STRUCT
	(* -----=== Byte 02 ===----- *)
	bFeederReq					:BIT;			//	Fuji adaagolóba menne a robot
	bPositioner1Req				:BIT;			//	Tájoló 1-be  menne a robot
	bPositioner2Req				:BIT;			//	Tájoló 2-be  menne a robot
	bFixtureAreaReq				:BIT;			//	PCB ülék fölé menne a robot
	bPositioner1OpenReq			:BIT;			//	Tájoló 1 nyitás kérés
	bPositioner2OpenReq			:BIT;			//	Tájoló 2 nyitás kérés
	{attribute 'hide'}
	_reserved_02_7				:BIT;			// Tartalék 02.07	
	{attribute 'hide'}
	_reserved_02_8				:BIT;			// Tartalék 02.08	
END_STRUCT
END_TYPE

// ---- POUs/Temp/Fanuc/ST_Fanuc_Handshake_Out.TcDUT
TYPE ST_Fanuc_Handshake_Out :
STRUCT
	(* -----=== Byte 03 ===----- *)
	bFeederEnable				:BIT;			//	Fuji adaagolóba mehet a robot
	bPositioner1Enable			:BIT;			//	Tájoló 1-be  mehet a robot
	bPositioner2Enable			:BIT;			//	Tájoló 2-be  mehet a robot
	bFixtureAreaEnable			:BIT;			//	PCB ülék fölé mehet a robot
	bPositioner1Open			:BIT;			//	Tájoló 1 nyitva
	bPositioner2Open			:BIT;			//	Tájoló 2 nyitva
	{attribute 'hide'}
	_reserved_03_7				:BIT;			// Tartalék 03.07	
	{attribute 'hide'}
	_reserved_03_8				:BIT;			// Tartalék 03.08	
END_STRUCT
END_TYPE

// ---- POUs/Temp/Fanuc/ST_Fanuc_In.TcDUT
TYPE ST_Fanuc_In :
STRUCT
	stCtrl					:ST_Fanuc_Control_In;
	stHandShake				:ST_Fanuc_HandShake_In;
	stArea					:ST_Fanuc_Area_In;
	stDIO					:ST_Fanuc_DIO_In;
	stAlarm					:ST_Fanuc_Alarm_In;
	stData					:ST_Fanuc_Data_In;
	stProg					:ST_Fanuc_Prog_In;
	stEmergency				:ST_Fanuc_Emergency_In;
END_STRUCT
END_TYPE

// ---- POUs/Temp/Fanuc/ST_Fanuc_ManPos.TcDUT
TYPE ST_Fanuc_ManPos :
STRUCT
	nPosX				:REAL;
	nPosY				:REAL;
	nPosR				:REAL;
END_STRUCT
END_TYPE

// ---- POUs/Temp/Fanuc/ST_Fanuc_Out.TcDUT
TYPE ST_Fanuc_Out :
STRUCT
	stCtrl					:ST_Fanuc_Control_Out;
	stHandShake				:ST_Fanuc_Handshake_Out;
	stPress					:ST_Fanuc_Press_Out;
	{attribute 'hide'}
	_reserved_05			:BYTE;						// Tartalék 05	
	stAlarm					:ST_Fanuc_Alarm_Out;
	stData					:ST_Fanuc_Data_Out;
	{attribute 'hide'}
	_reserved_13			:BYTE;						// Tartalék 13	
	stProg					:ST_Fanuc_Prog_Out;
END_STRUCT
END_TYPE

// ---- POUs/Temp/Fanuc/ST_Fanuc_Press_Out.TcDUT
TYPE ST_Fanuc_Press_Out :
STRUCT
	(* -----=== Byte 04 ===----- *)
	bWindow_1_Ok				:BIT;			//	Préselésifolyamat 1. ablak
	bWindow_2_Ok				:BIT;			//	Préselésifolyamat 2. ablak
	bWindow_3_Ok				:BIT;			//	Préselésifolyamat 3. ablak
	bWindow_4_Ok				:BIT;			//	Préselésifolyamat 4. ablak
	bWindow_5_Ok				:BIT;			//	Préselésifolyamat 5. ablak
	bWindow_6_Ok				:BIT;			//	Préselésifolyamat 6. ablak
	bWindow_7_Ok				:BIT;			//	Préselésifolyamat 7. ablak
	bWindow_8_Ok				:BIT;			//	Préselésifolyamat 8. ablak
END_STRUCT
END_TYPE

// ---- POUs/Temp/Fanuc/ST_Fanuc_Prog_In.TcDUT
TYPE ST_Fanuc_Prog_In :
STRUCT
	(* -----=== Byte 13 ===----- *)
	nActProg					:BYTE;			//	Aktuális program
	(* -----=== Byte 14 ===----- *)
	nActPoint					:BYTE;			//	Aktuális pont
END_STRUCT
END_TYPE

// ---- POUs/Temp/Fanuc/ST_Fanuc_Prog_Out.TcDUT
TYPE ST_Fanuc_Prog_Out :
STRUCT
	(* -----=== Byte 14 ===----- *)
	nType						:BYTE;			//	Típus kiválasztás
	(* -----=== Byte 15 ===----- *)
	nMode						:BYTE;			//	Üzemmód kiválasztás			Nincs használva
	(* -----=== Byte 16 ===----- *)
	nProgNr						:BYTE;			//	Mozgási program kiválasztás
END_STRUCT
END_TYPE

// ---- POUs/Temp/Fanuc/U_Fanuc_In.TcDUT
TYPE U_Fanuc_In :
UNION
	aFanuc_In		AT %I*	:ARRAY [1..16] OF BYTE;
	stFanucIn				:ST_Fanuc_In;
END_UNION
END_TYPE

// ---- POUs/Temp/Fanuc/U_Fanuc_Out.TcDUT
TYPE U_Fanuc_Out :
UNION
	aFanuc_Out		AT %Q*	:ARRAY [1..16] OF BYTE;
	stFanucOut				:ST_Fanuc_Out;
END_UNION
END_TYPE

// ---- GVLs/GVL_Ads.TcGVL
//{attribute 'qualified_only'}
VAR_GLOBAL
	OPC_UA_CNC1					: OPC_CNC_Data_Collection;	
	OPC_UA_CNC2					: OPC_CNC_Data_Collection;	
	OPC_UA_CNC3					: OPC_CNC_Data_Collection;	
	OPC_UA_CNC4					: OPC_CNC_Data_Collection;	
	OPC_UA_CNC5					: OPC_CNC_Data_Collection;	
END_VAR

// ---- GVLs/GVL_CNC1.TcGVL
VAR_GLOBAL
		stDutData_Cnc1					: ST_Dut_Data;
END_VAR

// ---- GVLs/GVL_CNC2.TcGVL
VAR_GLOBAL
		stDutData_Cnc2					: ST_Dut_Data;
END_VAR

// ---- GVLs/GVL_CNC3.TcGVL
VAR_GLOBAL
		stDutData_Cnc3					: ST_Dut_Data;
END_VAR

// ---- GVLs/GVL_Constant.TcGVL
VAR_GLOBAL CONSTANT
	nNbrOfAlarms				:BYTE := 40;
	cDarkBlue	:UDINT := 16#002A20A8;
	cTorquise	:UDINT := 16#007DD0D9;
	
	
	cBlack 		:UDINT := 16#00000000;
	cRed 		:UDINT := 16#008F0000;
	cOrange		:UDINT := 16#000F3200;
	cYellow		:UDINT := 16#000F0F00;
	cGreen 		:UDINT := 16#00000F00;
	cBlue 		:UDINT := 16#00000020;
	cIndigo		:UDINT := 16#0064005A;
	cViolet		:UDINT := 16#00C80064;
	cWhite 		:UDINT := 16#000F0F0F;
END_VAR

// ---- GVLs/GVL_ConveyorSystem.TcGVL
VAR_GLOBAL
	{attribute 'TcLinkTo' := 'TIIB(74)^Module 2 (CPI: 16 Byte I/0 Byte O)^Inputs^Input 0'}
	i_stSensorHub_0 AT %I* : ST_CPI_Module;					// S334
	{attribute 'TcLinkTo' := 'TIIB(74)^Module 2 (CPI: 16 Byte I/0 Byte O)^Inputs^Input 1'}
	i_stSensorHub_1 AT %I* : ST_CPI_Module;					// S314
	{attribute 'TcLinkTo' := 'TIIB(74)^Module 2 (CPI: 16 Byte I/0 Byte O)^Inputs^Input 2'}
	i_stSensorHub_2 AT %I* : ST_CPI_Module;					// S324
	{attribute 'TcLinkTo' := 'TIIB(74)^Module 2 (CPI: 16 Byte I/0 Byte O)^Inputs^Input 3'}
	i_stSensorHub_3 AT %I* : ST_CPI_Module;					// S344
	{attribute 'TcLinkTo' := 'TIIB(74)^Module 2 (CPI: 16 Byte I/0 Byte O)^Inputs^Input 4'}
	i_stSensorHub_4 AT %I* : ST_CPI_Module;					// S352
	{attribute 'TcLinkTo' := 'TIIB(74)^Module 2 (CPI: 16 Byte I/0 Byte O)^Inputs^Input 5'}
	i_stSensorHub_5 AT %I* : ST_CPI_Module;					// S313
	{attribute 'TcLinkTo' := 'TIIB(74)^Module 2 (CPI: 16 Byte I/0 Byte O)^Inputs^Input 6'}
	i_stSensorHub_6 AT %I* : ST_CPI_Module;					// S312
	{attribute 'TcLinkTo' := 'TIIB(74)^Module 2 (CPI: 16 Byte I/0 Byte O)^Inputs^Input 7'}
	i_stSensorHub_7 AT %I* : ST_CPI_Module;					// S311
	{attribute 'TcLinkTo' := 'TIIB(74)^Module 2 (CPI: 16 Byte I/0 Byte O)^Inputs^Input 8'}
	i_stSensorHub_8 AT %I* : ST_CPI_Module;					// S323
	{attribute 'TcLinkTo' := 'TIIB(74)^Module 2 (CPI: 16 Byte I/0 Byte O)^Inputs^Input 9'}
	i_stSensorHub_9 AT %I* : ST_CPI_Module;					// S351
	{attribute 'TcLinkTo' := 'TIIB(74)^Module 2 (CPI: 16 Byte I/0 Byte O)^Inputs^Input 10'}
	i_stSensorHub_10 AT %I* : ST_CPI_Module;				// S321
	{attribute 'TcLinkTo' := 'TIIB(74)^Module 2 (CPI: 16 Byte I/0 Byte O)^Inputs^Input 11'}
	i_stSensorHub_11 AT %I* : ST_CPI_Module;				// S322
	{attribute 'TcLinkTo' := 'TIIB(74)^Module 2 (CPI: 16 Byte I/0 Byte O)^Inputs^Input 12'}
	i_stSensorHub_12 AT %I* : ST_CPI_Module;				// S343
	{attribute 'TcLinkTo' := 'TIIB(74)^Module 2 (CPI: 16 Byte I/0 Byte O)^Inputs^Input 13'}
	i_stSensorHub_13 AT %I* : ST_CPI_Module;				// S333
	{attribute 'TcLinkTo' := 'TIIB(74)^Module 2 (CPI: 16 Byte I/0 Byte O)^Inputs^Input 14'}
	i_stSensorHub_14 AT %I* : ST_CPI_Module;				// S331
	{attribute 'TcLinkTo' := 'TIIB(74)^Module 2 (CPI: 16 Byte I/0 Byte O)^Inputs^Input 15'}
	i_stSensorHub_15 AT %I* : ST_CPI_Module;				// S332
	{attribute 'TcLinkTo' := 'TIIB(74)^Module 3 (CPI: 4 Byte I/0 Byte O)^Inputs^Input 0'}
	i_stSensorHub_16 AT %I* : ST_CPI_Module;				// S342
	{attribute 'TcLinkTo' := 'TIIB(74)^Module 3 (CPI: 4 Byte I/0 Byte O)^Inputs^Input 1'}
	i_stSensorHub_17 AT %I* : ST_CPI_Module;				// S341
	{attribute 'TcLinkTo' := 'TIIB(74)^Module 3 (CPI: 4 Byte I/0 Byte O)^Inputs^Input 2'}
	i_stSensorHub_18 AT %I* : ST_CPI_Module;			// Not included
	{attribute 'TcLinkTo' := 'TIIB(74)^Module 3 (CPI: 4 Byte I/0 Byte O)^Inputs^Input 3'}
	i_stSensorHub_19 AT %I* : ST_CPI_Module;			// Not included

(* Kiemelők *)	
	{attribute 'TcLinkTo' := 'TIIB(74)^Module 4 (MPA1G VMPA1-FB-EMG-8 [8DO])^Outputs^Output 0'}
	q_bZ1_14 AT %Q* : BOOL;
	{attribute 'TcLinkTo' := 'TIIB(74)^Module 4 (MPA1G VMPA1-FB-EMG-8 [8DO])^Outputs^Output 1'}
	q_bZ1_12 AT %Q* : BOOL;
	
	{attribute 'TcLinkTo' := 'TIIB(74)^Module 4 (MPA1G VMPA1-FB-EMG-8 [8DO])^Outputs^Output 2'}
	q_bZ2_14 AT %Q* : BOOL;
	{attribute 'TcLinkTo' := 'TIIB(74)^Module 4 (MPA1G VMPA1-FB-EMG-8 [8DO])^Outputs^Output 3'}
	q_bZ2_12 AT %Q* : BOOL;
	
	{attribute 'TcLinkTo' := 'TIIB(74)^Module 4 (MPA1G VMPA1-FB-EMG-8 [8DO])^Outputs^Output 4'}
	q_bZ3_14 AT %Q* : BOOL;
	{attribute 'TcLinkTo' := 'TIIB(74)^Module 4 (MPA1G VMPA1-FB-EMG-8 [8DO])^Outputs^Output 5'}
	q_bZ3_12 AT %Q* : BOOL;
	
	{attribute 'TcLinkTo' := 'TIIB(74)^Module 4 (MPA1G VMPA1-FB-EMG-8 [8DO])^Outputs^Output 6'}
	q_bZ4_14 AT %Q* : BOOL;
	{attribute 'TcLinkTo' := 'TIIB(74)^Module 4 (MPA1G VMPA1-FB-EMG-8 [8DO])^Outputs^Output 7'}
	q_bZ4_12 AT %Q* : BOOL;
	
	{attribute 'TcLinkTo' := 'TIIB(74)^Module 5 (MPA1G VMPA1-FB-EMG-8 [8DO])^Outputs^Output 0'}
	q_bZ5_14 AT %Q* : BOOL;
	{attribute 'TcLinkTo' := 'TIIB(74)^Module 5 (MPA1G VMPA1-FB-EMG-8 [8DO])^Outputs^Output 1'}
	q_bZ5_12 AT %Q* : BOOL;
	
	{attribute 'TcLinkTo' := 'TIIB(74)^Module 5 (MPA1G VMPA1-FB-EMG-8 [8DO])^Outputs^Output 2'}
	q_bZ6_14 AT %Q* : BOOL;
	{attribute 'TcLinkTo' := 'TIIB(74)^Module 5 (MPA1G VMPA1-FB-EMG-8 [8DO])^Outputs^Output 3'}
	q_bZ6_12 AT %Q* : BOOL;

(* Megfogók *)	
	{attribute 'TcLinkTo' := 'TIIB(74)^Module 5 (MPA1G VMPA1-FB-EMG-8 [8DO])^Outputs^Output 4'}
	q_bZ7_14 AT %Q* : BOOL;
	{attribute 'TcLinkTo' := 'TIIB(74)^Module 5 (MPA1G VMPA1-FB-EMG-8 [8DO])^Outputs^Output 5'}
	q_bZ7_12 AT %Q* : BOOL;

	{attribute 'TcLinkTo' := 'TIIB(74)^Module 5 (MPA1G VMPA1-FB-EMG-8 [8DO])^Outputs^Output 6'}
	q_bZ8_14 AT %Q* : BOOL;
	{attribute 'TcLinkTo' := 'TIIB(74)^Module 5 (MPA1G VMPA1-FB-EMG-8 [8DO])^Outputs^Output 7'}
	q_bZ8_12 AT %Q* : BOOL;

	{attribute 'TcLinkTo' := 'TIIB(74)^Module 6 (MPA1G VMPA1-FB-EMG-8 [8DO])^Outputs^Output 0'}
	q_bZ9_14 AT %Q* : BOOL;
	{attribute 'TcLinkTo' := 'TIIB(74)^Module 6 (MPA1G VMPA1-FB-EMG-8 [8DO])^Outputs^Output 1'}
	q_bZ9_12 AT %Q* : BOOL;

	{attribute 'TcLinkTo' := 'TIIB(74)^Module 6 (MPA1G VMPA1-FB-EMG-8 [8DO])^Outputs^Output 2'}
	q_bZ10_14 AT %Q* : BOOL;
	{attribute 'TcLinkTo' := 'TIIB(74)^Module 6 (MPA1G VMPA1-FB-EMG-8 [8DO])^Outputs^Output 3'}
	q_bZ10_12 AT %Q* : BOOL;

	{attribute 'TcLinkTo' := 'TIIB(74)^Module 6 (MPA1G VMPA1-FB-EMG-8 [8DO])^Outputs^Output 4'}
	q_bZ11_14 AT %Q* : BOOL;
	{attribute 'TcLinkTo' := 'TIIB(74)^Module 6 (MPA1G VMPA1-FB-EMG-8 [8DO])^Outputs^Output 5'}
	q_bZ11_12 AT %Q* : BOOL;

	{attribute 'TcLinkTo' := 'TIIB(74)^Module 6 (MPA1G VMPA1-FB-EMG-8 [8DO])^Outputs^Output 6'}
	q_bZ12_14 AT %Q* : BOOL;
	{attribute 'TcLinkTo' := 'TIIB(74)^Module 6 (MPA1G VMPA1-FB-EMG-8 [8DO])^Outputs^Output 7'}
	q_bZ12_12 AT %Q* : BOOL;
	
	{attribute 'TcLinkTo' := 'TIIB(74)^Module 7 (MPA1G VMPA1-FB-EMG-8 [8DO])^Outputs^Output 0'}
	q_bZ13_14 AT %Q* : BOOL;
	{attribute 'TcLinkTo' := 'TIIB(74)^Module 7 (MPA1G VMPA1-FB-EMG-8 [8DO])^Outputs^Output 1'}
	q_bZ13_12 AT %Q* : BOOL;
	
	{attribute 'TcLinkTo' := 'TIIB(74)^Module 7 (MPA1G VMPA1-FB-EMG-8 [8DO])^Outputs^Output 2'}
	q_bZ14_14 AT %Q* : BOOL;
	{attribute 'TcLinkTo' := 'TIIB(74)^Module 7 (MPA1G VMPA1-FB-EMG-8 [8DO])^Outputs^Output 3'}
	q_bZ14_12 AT %Q* : BOOL;
	
	{attribute 'TcLinkTo' := 'TIIB(74)^Module 7 (MPA1G VMPA1-FB-EMG-8 [8DO])^Outputs^Output 4'}
	q_bZ15_14 AT %Q* : BOOL;
	{attribute 'TcLinkTo' := 'TIIB(74)^Module 7 (MPA1G VMPA1-FB-EMG-8 [8DO])^Outputs^Output 5'}
	q_bZ15_12 AT %Q* : BOOL;
	
	{attribute 'TcLinkTo' := 'TIIB(74)^Module 7 (MPA1G VMPA1-FB-EMG-8 [8DO])^Outputs^Output 6'}
	q_bZ16_14 AT %Q* : BOOL;
	{attribute 'TcLinkTo' := 'TIIB(74)^Module 7 (MPA1G VMPA1-FB-EMG-8 [8DO])^Outputs^Output 7'}
	q_bZ16_12 AT %Q* : BOOL;
	
	{attribute 'TcLinkTo' := 'TIIB(74)^Module 8 (MPA1G VMPA1-FB-EMG-8 [8DO])^Outputs^Output 0'}
	q_bZ17_14 AT %Q* : BOOL;
	{attribute 'TcLinkTo' := 'TIIB(74)^Module 8 (MPA1G VMPA1-FB-EMG-8 [8DO])^Outputs^Output 1'}
	q_bZ17_12 AT %Q* : BOOL;
	
	{attribute 'TcLinkTo' := 'TIIB(74)^Module 8 (MPA1G VMPA1-FB-EMG-8 [8DO])^Outputs^Output 2'}
	q_bZ18_14 AT %Q* : BOOL;
	{attribute 'TcLinkTo' := 'TIIB(74)^Module 8 (MPA1G VMPA1-FB-EMG-8 [8DO])^Outputs^Output 3'}
	q_bZ18_12 AT %Q* : BOOL;
	
	{attribute 'TcLinkTo' := 'TIIB(74)^Module 8 (MPA1G VMPA1-FB-EMG-8 [8DO])^Outputs^Output 4'}
	q_bZ19_14 AT %Q* : BOOL;
	{attribute 'TcLinkTo' := 'TIIB(74)^Module 8 (MPA1G VMPA1-FB-EMG-8 [8DO])^Outputs^Output 5'}
	q_bZ19_12 AT %Q* : BOOL;
	
	{attribute 'TcLinkTo' := 'TIIB(74)^Module 8 (MPA1G VMPA1-FB-EMG-8 [8DO])^Outputs^Output 6'}
	q_bZ20_14 AT %Q* : BOOL;
	{attribute 'TcLinkTo' := 'TIIB(74)^Module 8 (MPA1G VMPA1-FB-EMG-8 [8DO])^Outputs^Output 7'}
	q_bZ20_12 AT %Q* : BOOL;
	
	{attribute 'TcLinkTo' := 'TIIB(74)^Module 9 (MPA1G VMPA1-FB-EMG-8 [8DO])^Outputs^Output 0'}
	q_bZ21_14 AT %Q* : BOOL;
	{attribute 'TcLinkTo' := 'TIIB(74)^Module 9 (MPA1G VMPA1-FB-EMG-8 [8DO])^Outputs^Output 1'}
	q_bZ21_12 AT %Q* : BOOL;
	
	{attribute 'TcLinkTo' := 'TIIB(74)^Module 9 (MPA1G VMPA1-FB-EMG-8 [8DO])^Outputs^Output 3'}
	q_bS1 AT %Q* : BOOL;
	{attribute 'TcLinkTo' := 'TIIB(74)^Module 9 (MPA1G VMPA1-FB-EMG-8 [8DO])^Outputs^Output 2'}
	q_bS2 AT %Q* : BOOL;
	{attribute 'TcLinkTo' := 'TIIB(74)^Module 9 (MPA1G VMPA1-FB-EMG-8 [8DO])^Outputs^Output 5'}
	q_bS3 AT %Q* : BOOL;
	{attribute 'TcLinkTo' := 'TIIB(74)^Module 9 (MPA1G VMPA1-FB-EMG-8 [8DO])^Outputs^Output 4'}
	q_bS4 AT %Q* : BOOL;
	{attribute 'TcLinkTo' := 'TIIB(74)^Module 9 (MPA1G VMPA1-FB-EMG-8 [8DO])^Outputs^Output 7'}
	q_bS5 AT %Q* : BOOL;
	{attribute 'TcLinkTo' := 'TIIB(74)^Module 9 (MPA1G VMPA1-FB-EMG-8 [8DO])^Outputs^Output 6'}
	q_bS6 AT %Q* : BOOL;
	{attribute 'TcLinkTo' := 'TIIB(74)^Module 10 (MPA1G VMPA1-FB-EMG-8 [8DO])^Outputs^Output 1'}
	q_bS7 AT %Q* : BOOL;
	{attribute 'TcLinkTo' := 'TIIB(74)^Module 10 (MPA1G VMPA1-FB-EMG-8 [8DO])^Outputs^Output 0'}
	q_bS8 AT %Q* : BOOL;
	{attribute 'TcLinkTo' := 'TIIB(74)^Module 10 (MPA1G VMPA1-FB-EMG-8 [8DO])^Outputs^Output 3'}
	q_bS9 AT %Q* : BOOL;
	{attribute 'TcLinkTo' := 'TIIB(74)^Module 10 (MPA1G VMPA1-FB-EMG-8 [8DO])^Outputs^Output 2'}
	q_bS10 AT %Q* : BOOL;
	{attribute 'TcLinkTo' := 'TIIB(74)^Module 10 (MPA1G VMPA1-FB-EMG-8 [8DO])^Outputs^Output 5'}
	q_bS11 AT %Q* : BOOL;
	{attribute 'TcLinkTo' := 'TIIB(74)^Module 10 (MPA1G VMPA1-FB-EMG-8 [8DO])^Outputs^Output 4'}
	q_bS12 AT %Q* : BOOL;
	{attribute 'TcLinkTo' := 'TIIB(74)^Module 10 (MPA1G VMPA1-FB-EMG-8 [8DO])^Outputs^Output 7'}
	q_bS13 AT %Q* : BOOL;
	{attribute 'TcLinkTo' := 'TIIB(74)^Module 10 (MPA1G VMPA1-FB-EMG-8 [8DO])^Outputs^Output 6'}
	q_bS14 AT %Q* : BOOL;
	{attribute 'TcLinkTo' := 'TIIB(74)^Module 11 (MPA1G VMPA1-FB-EMG-8 [8DO])^Outputs^Output 1'}
	q_bS15 AT %Q* : BOOL;
	{attribute 'TcLinkTo' := 'TIIB(74)^Module 11 (MPA1G VMPA1-FB-EMG-8 [8DO])^Outputs^Output 0'}
	q_bS16 AT %Q* : BOOL;
	{attribute 'TcLinkTo' := 'TIIB(74)^Module 11 (MPA1G VMPA1-FB-EMG-8 [8DO])^Outputs^Output 3'}
	q_bS17 AT %Q* : BOOL;
	{attribute 'TcLinkTo' := 'TIIB(74)^Module 11 (MPA1G VMPA1-FB-EMG-8 [8DO])^Outputs^Output 2'}
	q_bS18 AT %Q* : BOOL;
	{attribute 'TcLinkTo' := 'TIIB(74)^Module 11 (MPA1G VMPA1-FB-EMG-8 [8DO])^Outputs^Output 5'}
	q_bS19 AT %Q* : BOOL;
	{attribute 'TcLinkTo' := 'TIIB(74)^Module 11 (MPA1G VMPA1-FB-EMG-8 [8DO])^Outputs^Output 4'}
	q_bS20 AT %Q* : BOOL;
	{attribute 'TcLinkTo' := 'TIIB(74)^Module 11 (MPA1G VMPA1-FB-EMG-8 [8DO])^Outputs^Output 7'}
	q_bS21 AT %Q* : BOOL;
	{attribute 'TcLinkTo' := 'TIIB(74)^Module 11 (MPA1G VMPA1-FB-EMG-8 [8DO])^Outputs^Output 6'}
	q_bS22 AT %Q* : BOOL;
	{attribute 'TcLinkTo' := 'TIIB(74)^Module 12 (MPA1G VMPA1-FB-EMG-8 [8DO])^Outputs^Output 1'}
	q_bS23 AT %Q* : BOOL;
	{attribute 'TcLinkTo' := 'TIIB(74)^Module 12 (MPA1G VMPA1-FB-EMG-8 [8DO])^Outputs^Output 0'}
	q_bS24 AT %Q* : BOOL;
	{attribute 'TcLinkTo' := 'TIIB(74)^Module 12 (MPA1G VMPA1-FB-EMG-8 [8DO])^Outputs^Output 3'}
	q_bS25 AT %Q* : BOOL;
	{attribute 'TcLinkTo' := 'TIIB(74)^Module 12 (MPA1G VMPA1-FB-EMG-8 [8DO])^Outputs^Output 2'}
	q_bS26 AT %Q* : BOOL;
	{attribute 'TcLinkTo' := 'TIIB(74)^Module 12 (MPA1G VMPA1-FB-EMG-8 [8DO])^Outputs^Output 5'}
	q_bS27 AT %Q* : BOOL;
	{attribute 'TcLinkTo' := 'TIIB(74)^Module 12 (MPA1G VMPA1-FB-EMG-8 [8DO])^Outputs^Output 4'}
	q_bS28 AT %Q* : BOOL;
	{attribute 'TcLinkTo' := 'TIIB(74)^Module 12 (MPA1G VMPA1-FB-EMG-8 [8DO])^Outputs^Output 7'}
	q_bS29 AT %Q* : BOOL;
	{attribute 'TcLinkTo' := 'TIIB(74)^Module 12 (MPA1G VMPA1-FB-EMG-8 [8DO])^Outputs^Output 6'}
	q_bS30 AT %Q* : BOOL;
	{attribute 'TcLinkTo' := 'TIIB(74)^Module 13 (MPA1G VMPA1-FB-EMG-8 [8DO])^Outputs^Output 1'}
	q_bS31 AT %Q* : BOOL;
	{attribute 'TcLinkTo' := 'TIIB(74)^Module 13 (MPA1G VMPA1-FB-EMG-8 [8DO])^Outputs^Output 0'}
	q_bS32 AT %Q* : BOOL;
END_VAR
VAR_GLOBAL (* Stoppers *)
	fbS1 : FB_Stopper;
	fbS2 : FB_Stopper;
	fbS3 : FB_Stopper;
	fbS4 : FB_Stopper;
	fbS5 : FB_Stopper;
	fbS6 : FB_Stopper;
	fbS7 : FB_Stopper;
	fbS8 : FB_Stopper2;
	fbS9 : FB_Stopper2;
	fbS10 : FB_Stopper2;
	fbS11 : FB_Stopper2;
	fbS12 : FB_Stopper2;
	fbS13 : FB_Stopper;
	fbS14 : FB_Stopper;
	fbS15 : FB_Stopper2;
	fbS16 : FB_Stopper2;
	fbS17 : FB_Stopper;
	fbS18 : FB_Stopper2;
	fbS19 : FB_Stopper;
	fbS20 : FB_Stopper2;
	fbS21 : FB_Stopper2;
	fbS22 : FB_Stopper;
	fbS23 : FB_Stopper;
	fbS24 : FB_Stopper2;
	fbS25 : FB_Stopper2;
	fbS26 : FB_Stopper2;
	fbS27 : FB_Stopper2;
	fbS28 : FB_Stopper; // 28 hol faszom sem tudja
	fbS29 : FB_Stopper;
	fbS30 : FB_Stopper2;
	fbS31 : FB_Stopper2;
	fbS32 : FB_Stopper;
END_VAR
VAR_GLOBAL (* Cylinders *)
	fbZ1 : FB_Bistabil;
	fbZ2 : FB_Bistabil;
	fbZ3 : FB_Bistabil;
	fbZ4 : FB_Bistabil;
	fbZ5 : FB_Bistabil;
	fbZ6 : FB_Bistabil;
	fbZ7 : FB_Bistabil;
	fbZ8 : FB_Bistabil;
	fbZ9 : FB_Bistabil;
	fbZ10 : FB_Bistabil;
	fbZ11 : FB_Bistabil;
	fbZ12 : FB_Bistabil;
	fbZ13 : FB_Bistabil;
	fbZ14 : FB_Bistabil;
	fbZ15 : FB_Bistabil;
	fbZ16 : FB_Bistabil;
	fbZ17 : FB_Bistabil;
	fbZ18 : FB_Bistabil;
	fbZ19 : FB_Bistabil;
	fbZ20 : FB_Bistabil;
	fbZ21 : FB_Bistabil;
END_VAR
VAR_GLOBAL	(* Conveyors *)
	fbConveyor_1		: FB_Conveyor;
	fbConveyor_2		: FB_Conveyor;
	fbConveyor_3		: FB_Conveyor;
	fbConveyor_4		: FB_Conveyor;
	fbConveyor_5		: FB_Conveyor;
	fbConveyor_6		: FB_Conveyor;
	fbConveyor_7		: FB_Conveyor;
	fbConveyor_8		: FB_Conveyor;
	fbConveyor_9		: FB_Conveyor;
	fbConveyor_10		: FB_Conveyor;
	fbConveyor_11		: FB_Conveyor;
END_VAR
VAR_GLOBAL
	fbLift_1A			: FB_Lift;
	fbLift_1B			: FB_Lift;
	fbLift_2A			: FB_Lift;
	fbLift_2B			: FB_Lift;
	fbLift_3A			: FB_Lift;
	fbLift_3B			: FB_Lift;
END_VAR
VAR_GLOBAL
	fbRouter_CNC1_puffer	: FB_Router;
	fbRouter_CNC2_puffer	: FB_Router;
	fbRouter_CNC3_puffer	: FB_Router;

END_VAR

// ---- GVLs/GVL_IO.TcGVL
VAR_GLOBAL
(**************************************************Inputs*********************************************************)	
	// 1.x
	// Satuzó 1-7
	{attribute 'TcLinkTo' := 'TIIB(82)^Channel 1^Input'} 
	i_bVisePos1InBtn			AT %I*	:BOOL;		// Satu be 1-7
	{attribute 'TcLinkTo' := 'TIIB(82)^Channel 2^Input'}
	i_bVisePos1RequestBtn		AT %I*	:BOOL;		// Satu kérés 1-7
	{attribute 'TcLinkTo' := 'TIIB(82)^Channel 3^Input'}
	i_bVisePos1CleanBtn			AT %I*	:BOOL;		// Satu tisztítás 1-7
	{attribute 'TcLinkTo' := 'TIIB(82)^Channel 4^Input'}
	i_bVisePos1ErrorAckBtn		AT %I*	:BOOL;		// Satu hibanyugta 1-7

	// Satuzó 8-14
	{attribute 'TcLinkTo' := 'TIIB(82)^Channel 5^Input'}
	i_bVisePos2InBtn			AT %I*	:BOOL;		// Satu be 8-14
	{attribute 'TcLinkTo' := 'TIIB(82)^Channel 6^Input'}
	i_bVisePos2RequestBtn		AT %I*	:BOOL;		// Satu kérés 8-14
	{attribute 'TcLinkTo' := 'TIIB(82)^Channel 7^Input'}
	i_bVisePos2CleanBtn			AT %I*	:BOOL;		// Satu tisztítás 8-14
	{attribute 'TcLinkTo' := 'TIIB(82)^Channel 8^Input'}
	i_bVisePos2ErrorAckBtn		AT %I*	:BOOL;		// Satu hibanyugta 8-14
	
	{attribute 'TcLinkTo' := 'TIIB(82)^Channel 9^Input'}
	i_bAirPressureOk			AT %I*	:BOOL;		// Levegő nyomás OK
	{attribute 'TcLinkTo' := 'TIIB(82)^Channel 10^Input'}
	i_bCellAck					AT %I*	:BOOL;		// Satuzó ajtó zárás nyugtázás - kék gomb
	{attribute 'TcLinkTo' := 'TIIB(82)^Channel 11^Input'}
	i_bCaptron					AT %I*	:BOOL;		// Operator Captron
	
	// 2.x
	{attribute 'TcLinkTo' := 'TIIB(83)^Channel 1^Input'}
	i_bEMYStop1					AT %I*	:BOOL;		// Vészstop 1
	{attribute 'TcLinkTo' := 'TIIB(83)^Channel 2^Input'}
	i_bEMYStop2					AT %I*	:BOOL;		// Vészstop 2
	{attribute 'TcLinkTo' := 'TIIB(83)^Channel 3^Input'}
	i_bEMYStop3					AT %I*	:BOOL;		// Vészstop 3
	{attribute 'TcLinkTo' := 'TIIB(83)^Channel 4^Input'}
	i_bEMYStop4					AT %I*	:BOOL;		// Vészstop 4
	{attribute 'TcLinkTo' := 'TIIB(83)^Channel 5^Input'}
	i_bEMYStop5					AT %I*	:BOOL;		// Vészstop 5
	{attribute 'TcLinkTo' := 'TIIB(83)^Channel 6^Input'}
	i_bEMYStop6					AT %I*	:BOOL;		// Vészstop 6	
	{attribute 'TcLinkTo' := 'TIIB(83)^Channel 9^Input'}
	i_bDoorClosed				AT %I*	:BOOL;		// Ajtó nyitva/zárva
	{attribute 'TcLinkTo' := 'TIIB(83)^Channel 10^Input'}
	i_bMasterOn_CNC45					AT %I*	:BOOL;		// Vezérlés
	{attribute 'TcLinkTo' := 'TIIB(83)^Channel 11^Input'}
	i_bDoorRequest				AT %I*	:BOOL;		// Ajtó nyítás kérés

	
(**************************************************Outputs*********************************************************)
	{attribute 'TcLinkTo' := 'TIIB(84)^Channel 1^Output'}
	q_bMasterOnLED				AT %Q*	:BOOL;		// Vezérlés LED
	{attribute 'TcLinkTo' := 'TIIB(84)^Channel 2^Output'}
	q_bDoorRequestLED			AT %Q*	:BOOL;		// Ajtó nyítás kérés LED
	
	// Satuzó 1-7
	{attribute 'TcLinkTo' := 'TIIB(84)^Channel 3^Output'}
	q_bVise1InLED				AT %Q*	:BOOL;		// Satu be 1-7 LED
	{attribute 'TcLinkTo' := 'TIIB(84)^Channel 4^Output'}
	q_bVise1ReqestLED			AT %Q*	:BOOL;		// Satu kérés 1-7 LED
	{attribute 'TcLinkTo' := 'TIIB(84)^Channel 5^Output'}
	q_bVise1CleanLED			AT %Q*	:BOOL;		// Satu tisztítás 1-7 LED
	{attribute 'TcLinkTo' := 'TIIB(84)^Channel 6^Output'}
	q_bVise1ErrorAckLED 		AT %Q*	:BOOL;		// Satu hibanyugta 1-7 LED
	
	// Satuzó 8-14
	{attribute 'TcLinkTo' := 'TIIB(84)^Channel 7^Output'}
	q_bVise2InLED				AT %Q*	:BOOL;		// Satu be 8-14 LED
	{attribute 'TcLinkTo' := 'TIIB(84)^Channel 8^Output'}
	q_bVise2RequestLED			AT %Q*	:BOOL;		// Satu kérés 8-14 LED
	{attribute 'TcLinkTo' := 'TIIB(84)^Channel 9^Output'}
	q_bVise2CleanLED			AT %Q*	:BOOL;		// Satu tisztítás 8-14 LED
	{attribute 'TcLinkTo' := 'TIIB(84)^Channel 10^Output'}
	q_bVise2ErrorAckBtnLED		AT %Q*	:BOOL;		// Satu hibanyugta 8-14 LED
	
	{attribute 'TcLinkTo' := 'TIIB(84)^Channel 11^Output'}
	q_bDoorLock					AT %Q*	:BOOL;		// Ajtó zárás
	{attribute 'TcLinkTo' := 'TIIB(84)^Channel 12^Output'}
	q_bCellAckLED				AT %Q*	:BOOL;		// Satuzó ajtó zárás nyugtázás - kék gomb LED
	{attribute 'TcLinkTo' := 'TIIB(84)^Channel 13^Output'}
	q_bCaptronLED				AT %Q*	:BOOL;		// Operator Captron LED
	{attribute 'TcLinkTo' := 'TIIB(60)^InfoData^State'}
	i_nBusState					AT %I*	:uint;
	
(**************************************************Festo Inputs*********************************************************)	
	// Satuzó 1-7
 	{attribute 'TcLinkToOSO' := ' <0,8,0>TIIB(88)^Input^Inputs^Input 0;
    						 	  <8,8,0>TIIB(88)^Input^Inputs^Input 1;'}
	i_stViseStationSensors_1	AT %I*	:ST_Vise_Sensors;
	{attribute 'TcLinkToOSO' := '<0,8,0>TIIB(88)^Input^Inputs^Input 2;
								 <8,8,0>TIIB(88)^Input^Inputs^Input 3'}
	i_stViseStationSensors_2	AT %I*	:ST_Vise_Sensors;
	{attribute 'TcLinkToOSO' := '<0,8,0>TIIB(88)^Input^Inputs^Input 4;
								 <8,8,0>TIIB(88)^Input^Inputs^Input 5'}
	i_stViseStationSensors_3	AT %I*	:ST_Vise_Sensors;
	{attribute 'TcLinkToOSO' := ' <0,8,0>TIIB(88)^Input^Inputs^Input 6;
    						 	  <8,8,0>TIIB(88)^Input^Inputs^Input 7;'}
	i_stViseStationSensors_4	AT %I*	:ST_Vise_Sensors;
	{attribute 'TcLinkToOSO' := '<0,8,0>TIIB(88)^Input^Inputs^Input 8;
								 <8,8,0>TIIB(88)^Input^Inputs^Input 9'}
	i_stViseStationSensors_5	AT %I*	:ST_Vise_Sensors;
	{attribute 'TcLinkToOSO' := '<0,8,0>TIIB(88)^Input^Inputs^Input 10;
								 <8,8,0>TIIB(88)^Input^Inputs^Input 11'}
	i_stViseStationSensors_6	AT %I*	:ST_Vise_Sensors;
	{attribute 'TcLinkToOSO' := '<0,8,0>TIIB(88)^Input^Inputs^Input 12;
								 <8,8,0>TIIB(88)^Input^Inputs^Input 13'}
	i_stViseStationSensors_7	AT %I*	:ST_Vise_Sensors;
	
	// Satuzó 8-14
 	{attribute 'TcLinkToOSO' := ' <0,8,0>TIIB(89)^Input^Inputs^Input 0;
    						 	  <8,8,0>TIIB(89)^Input^Inputs^Input 1;'}
	i_stViseStationSensors_8	AT %I*	:ST_Vise_Sensors;
	{attribute 'TcLinkToOSO' := '<0,8,0>TIIB(89)^Input^Inputs^Input 2;
								 <8,8,0>TIIB(89)^Input^Inputs^Input 3'}
	i_stViseStationSensors_9	AT %I*	:ST_Vise_Sensors;
	{attribute 'TcLinkToOSO' := '<0,8,0>TIIB(89)^Input^Inputs^Input 4;
								 <8,8,0>TIIB(89)^Input^Inputs^Input 5'}
	i_stViseStationSensors_10	AT %I*	:ST_Vise_Sensors;
	{attribute 'TcLinkToOSO' := ' <0,8,0>TIIB(89)^Input^Inputs^Input 6;
    						 	  <8,8,0>TIIB(89)^Input^Inputs^Input 7;'}
	i_stViseStationSensors_11	AT %I*	:ST_Vise_Sensors;
	{attribute 'TcLinkToOSO' := '<0,8,0>TIIB(89)^Input^Inputs^Input 8;
								 <8,8,0>TIIB(89)^Input^Inputs^Input 9'}
	i_stViseStationSensors_12	AT %I*	:ST_Vise_Sensors;
	{attribute 'TcLinkToOSO' := '<0,8,0>TIIB(89)^Input^Inputs^Input 10;
								 <8,8,0>TIIB(89)^Input^Inputs^Input 11'}
	i_stViseStationSensors_13	AT %I*	:ST_Vise_Sensors;
	{attribute 'TcLinkToOSO' := '<0,8,0>TIIB(89)^Input^Inputs^Input 12;
								 <8,8,0>TIIB(89)^Input^Inputs^Input 13'}
	i_stViseStationSensors_14	AT %I*	:ST_Vise_Sensors;
END_VAR
VAR_GLOBAL
(**************************************************CNC45 Inputs*********************************************************)
	{attribute 'TcLinkTo' := 'TIIB(91)^Channel 1^Input'} 
	i_bCNC4_Door_Opened			AT %I*	:BOOL;
	{attribute 'TcLinkTo' := 'TIIB(91)^Channel 2^Input'} 
	i_bCNC4_Door_Closed			AT %I*	:BOOL;
	{attribute 'TcLinkTo' := 'TIIB(91)^Channel 3^Input'}
	i_bCNC4_Program_Ready		AT %I*	:BOOL;
	{attribute 'TcLinkTo' := 'TIIB(91)^Channel 4^Input'}
	i_bCNC4_Program_Run			AT %I*	:BOOL;
	{attribute 'TcLinkTo' := 'TIIB(91)^Channel 5^Input'}
	i_bCNC4_Program_End			AT %I*	:BOOL;
	{attribute 'TcLinkTo' := 'TIIB(91)^Channel 6^Input'}
	i_bCNC4_Error				AT %I*	:BOOL;
	{attribute 'TcLinkTo' := 'TIIB(91)^Channel 7^Input'}
	i_bCNC4_Robot_Mode			AT %I*	:BOOL;
	{attribute 'TcLinkTo' := 'TIIB(91)^Channel 8^Input'}
	i_bCNC4_M401_Req			AT %I*	:BOOL;
	{attribute 'TcLinkTo' := 'TIIB(91)^Channel 9^Input'}
	i_bCNC4_M402_Req			AT %I*	:BOOL;
	{attribute 'TcLinkTo' := 'TIIB(91)^Channel 10^Input'}
	i_bCNC4_M403_Req			AT %I*	:BOOL;
	{attribute 'TcLinkTo' := 'TIIB(91)^Channel 11^Input'}
	i_bCNC4_Door_HW_opened		AT %I*	:BOOL;
	
(**************************************************CNC45 Outputs*********************************************************)
	{attribute 'TcLinkTo' := 'TIIB(92)^Channel 1^Output'}
	q_bCNC4_Door_Open			AT %Q*	:BOOL;
	{attribute 'TcLinkTo' := 'TIIB(92)^Channel 2^Output'}
	q_bCNC4_Door_Close			AT %Q*	:BOOL;
	{attribute 'TcLinkTo' := 'TIIB(92)^Channel 3^Output'}
	q_bCNC4_Program_Start		AT %Q*	:BOOL;
	{attribute 'TcLinkTo' := 'TIIB(92)^Channel 4^Output'}
	q_bCNC4_M401_Ack			AT %Q*	:BOOL;
	{attribute 'TcLinkTo' := 'TIIB(92)^Channel 5^Output'}
	q_bCNC4_M402_Ack			AT %Q*	:BOOL;
	{attribute 'TcLinkTo' := 'TIIB(92)^Channel 6^Output'}
	q_bCNC4_M403_Ack			AT %Q*	:BOOL;
	
	{attribute 'TcLinkTo' := 'TIIB(92)^Channel 7^Output'}
	q_bCNC4_Fix_Vise			AT %Q*	:BOOL;
	{attribute 'TcLinkTo' := 'TIIB(92)^Channel 8^Output'}
	q_bCNC4_Release_Vise		AT %Q* 	:BOOL;
	{attribute 'TcLinkTo' := 'TIIB(92)^Channel 9^Output'}
	q_bCNC4_CleanTool			AT %Q* 	:BOOL;

END_VAR
VAR_GLOBAL
(**************************************************Inputs*********************************************************)	
	// I20.x
	// Main EK1100/1 (with safety plc)
	{attribute 'TcLinkTo' := 'TIIB(48)^Channel 1^Input'}
	i_bConveyor_1_Ok			AT %I*	:BOOL;		// Konvejor
	{attribute 'TcLinkTo' := 'TIIB(48)^Channel 2^Input'}
	i_bConveyor_2_Ok			AT %I*	:BOOL;		// Konvejor
	{attribute 'TcLinkTo' := 'TIIB(48)^Channel 3^Input'}
	i_bConveyor_3_Ok			AT %I*	:BOOL;		// Konvejor
	{attribute 'TcLinkTo' := 'TIIB(48)^Channel 4^Input'}
	i_bConveyor_4_Ok			AT %I*	:BOOL;		// Konvejor
	{attribute 'TcLinkTo' := 'TIIB(48)^Channel 5^Input'}
	i_bConveyor_5_Ok			AT %I*	:BOOL;		// Konvejor
	{attribute 'TcLinkTo' := 'TIIB(48)^Channel 6^Input'}
	i_bConveyor_6_Ok			AT %I*	:BOOL;		// Konvejor
	{attribute 'TcLinkTo' := 'TIIB(48)^Channel 7^Input'}
	i_bConveyor_7_Ok			AT %I*	:BOOL;		// Konvejor
	{attribute 'TcLinkTo' := 'TIIB(48)^Channel 8^Input'}
	i_bConveyor_8_Ok			AT %I*	:BOOL;		// Konvejor
	{attribute 'TcLinkTo' := 'TIIB(48)^Channel 9^Input'}
	i_bConveyor_9_Ok			AT %I*	:BOOL;		// Konvejor
	{attribute 'TcLinkTo' := 'TIIB(48)^Channel 10^Input'}
	i_bConveyor_10_Ok			AT %I*	:BOOL;		// Konvejor
	{attribute 'TcLinkTo' := 'TIIB(48)^Channel 11^Input'}
	i_bConveyor_11_Ok			AT %I*	:BOOL;		// Konvejor
	{attribute 'TcLinkTo' := 'TIIB(48)^Channel 12^Input'}
	i_bTerm48_Ch12				AT %I*	:BOOL;		// Konvejor
	{attribute 'TcLinkTo' := 'TIIB(48)^Channel 13^Input'}
	i_bTerm48_Ch13				AT %I*	:BOOL;		// Konvejor
	{attribute 'TcLinkTo' := 'TIIB(48)^Channel 14^Input'}
	i_bTerm48_Ch14				AT %I*	:BOOL;		// Konvejor
	{attribute 'TcLinkTo' := 'TIIB(48)^Channel 15^Input'}
	i_bTerm48_Ch15				AT %I*	:BOOL;		// Konvejor
	{attribute 'TcLinkTo' := 'TIIB(48)^Channel 16^Input'}
	i_bTerm48_Ch16				AT %I*	:BOOL;		// Konvejor
	
	// I21.x
	{attribute 'TcLinkTo' := 'TIIB(49)^Channel 1^Input'}
	i_bEMYStop10				AT %I*	:BOOL;		// Vészstop 10
	{attribute 'TcLinkTo' := 'TIIB(49)^Channel 2^Input'}
	i_bEMYStop11				AT %I*	:BOOL;		// Vészstop 11
	{attribute 'TcLinkTo' := 'TIIB(49)^Channel 3^Input'}
	i_bEMYStop12				AT %I*	:BOOL;		// Vészstop 12
	{attribute 'TcLinkTo' := 'TIIB(49)^Channel 4^Input'}
	i_bEMYStop13				AT %I*	:BOOL;		// Vészstop 13
	{attribute 'TcLinkTo' := 'TIIB(49)^Channel 5^Input'}
	i_bEMYStop14				AT %I*	:BOOL;		// Vészstop 14
	{attribute 'TcLinkTo' := 'TIIB(49)^Channel 6^Input'}
	i_bEMYStop15				AT %I*	:BOOL;		// Vészstop 15
	{attribute 'TcLinkTo' := 'TIIB(49)^Channel 7^Input'}
	i_bEMYStop16				AT %I*	:BOOL;		// Vészstop 16
	{attribute 'TcLinkTo' := 'TIIB(49)^Channel 8^Input'}
	i_bEMYStop17				AT %I*	:BOOL;		// Vészstop 17
	{attribute 'TcLinkTo' := 'TIIB(49)^Channel 9^Input'}
	i_bDoorClosed_Kardex		AT %I*	:BOOL;		// Ajtó nyitva/zárva
	{attribute 'TcLinkTo' := 'TIIB(49)^Channel 10^Input'}
	i_bMasterOn_Kardex			AT %I*	:BOOL;		// Vezérlés
	{attribute 'TcLinkTo' := 'TIIB(49)^Channel 11^Input'}
	i_bDoorRequest_Kardex		AT %I*	:BOOL;		// Ajtó nyítás kérés
	{attribute 'TcLinkTo' := 'TIIB(49)^Channel 12^Input'}
	i_bDoorClosed_Main			AT %I*	:BOOL;		// Ajtó nyitva/zárva
	{attribute 'TcLinkTo' := 'TIIB(49)^Channel 13^Input'}
	i_bMasterOn_Main			AT %I*	:BOOL;		// Vezérlés
	{attribute 'TcLinkTo' := 'TIIB(49)^Channel 14^Input'}
	i_bDoorRequest_Main			AT %I*	:BOOL;		// Ajtó nyítás kérés
	{attribute 'TcLinkTo' := 'TIIB(49)^Channel 15^Input'}
	i_bTerm49_Ch15				AT %I*	:BOOL;		// Konvejor
	{attribute 'TcLinkTo' := 'TIIB(49)^Channel 16^Input'}
	i_bTerm49_Ch16				AT %I*	:BOOL;		// Konvejor


	// I22.x
	{attribute 'TcLinkTo' := 'TIIB(50)^Channel 1^Input'} 
	i_bTest_01					AT %I*	:BOOL;		// Test 01
	{attribute 'TcLinkTo' := 'TIIB(50)^Channel 2^Input'}
	i_bErrorAckBtn_Main			AT %I*	:BOOL;		// Error Ack
	{attribute 'TcLinkTo' := 'TIIB(50)^Channel 3^Input'}
	i_bTest03					AT %I*	:BOOL;		// Test 03
//	{attribute 'TcLinkTo' := 'TIIB(50)^Channel 4^Input'}
//	i_bMasterOn_Main			AT %I*	:BOOL;		// Master On
	{attribute 'TcLinkTo' := 'TIIB(50)^Channel 5^Input'}
	i_bTest_Up					AT %I*	:BOOL;		// Master On
	{attribute 'TcLinkTo' := 'TIIB(50)^Channel 6^Input'}
	i_bTest_Stop				AT %I*	:BOOL;		// Master On
	{attribute 'TcLinkTo' := 'TIIB(50)^Channel 7^Input'}
	i_bTest_Down				AT %I*	:BOOL;		// Master On

(**************************************************Outputs*********************************************************)
	// Q20.x
	{attribute 'TcLinkTo' := 'TIIB(51)^Channel 1^Output'}
	q_bMasterOnLED_Kardex		AT %Q*	:BOOL;		// Vezérlés LED
	{attribute 'TcLinkTo' := 'TIIB(51)^Channel 2^Output'}
	q_bDoorRequestLED_Kardex	AT %Q*	:BOOL;		// Ajtó nyítás kérés LED
	{attribute 'TcLinkTo' := 'TIIB(51)^Channel 3^Output'}
	q_bMasterOnLED_Main			AT %Q*	:BOOL;		// Vezérlés LED
	{attribute 'TcLinkTo' := 'TIIB(51)^Channel 4^Output'}
	q_bDoorRequestLED_Main	AT %Q*	:BOOL;		// Ajtó nyítás kérés LED

	{attribute 'TcLinkTo' := 'TIIB(54)^Channel 1^Output'}
	q_bConveyor_1				AT %Q*	:BOOL;		// Konvejor
	{attribute 'TcLinkTo' := 'TIIB(54)^Channel 2^Output'}
	q_bConveyor_2				AT %Q*	:BOOL;		// Konvejor
	{attribute 'TcLinkTo' := 'TIIB(54)^Channel 3^Output'}
	q_bConveyor_3				AT %Q*	:BOOL;		// Konvejor
	{attribute 'TcLinkTo' := 'TIIB(54)^Channel 4^Output'}
	q_bConveyor_4				AT %Q*	:BOOL;		// Konvejor
	{attribute 'TcLinkTo' := 'TIIB(54)^Channel 5^Output'}
	q_bConveyor_5				AT %Q*	:BOOL;		// Konvejor
	{attribute 'TcLinkTo' := 'TIIB(54)^Channel 6^Output'}
	q_bConveyor_6				AT %Q*	:BOOL;		// Konvejor
	{attribute 'TcLinkTo' := 'TIIB(54)^Channel 7^Output'}
	q_bConveyor_7				AT %Q*	:BOOL;		// Konvejor
	{attribute 'TcLinkTo' := 'TIIB(54)^Channel 8^Output'}
	q_bConveyor_8				AT %Q*	:BOOL;		// Konvejor
	{attribute 'TcLinkTo' := 'TIIB(54)^Channel 9^Output'}
	q_bConveyor_9				AT %Q*	:BOOL;		// Konvejor
	{attribute 'TcLinkTo' := 'TIIB(54)^Channel 10^Output'}
	q_bConveyor_10				AT %Q*	:BOOL;		// Konvejor
	{attribute 'TcLinkTo' := 'TIIB(54)^Channel 11^Output'}
	q_bConveyor_11				AT %Q*	:BOOL;		// Konvejor

(**************************************************7Axis Fanuc*********************************************************)
	{attribute 'TcLinkTo' := '		.arrRaw[0]	:= TIIB(8)^Module 1 (IOL_I_2byte)^TxPDO^input byte 0;	
									.arrRaw[1] 	:= TIIB(8)^Module 1 (IOL_I_2byte)^TxPDO^input byte 1;
									.nState		:= TIIB(8)^IO-Link DeviceState Inputs^Status of IO-Link Port 1;'}
	fbGripperPos1				: FB_MPS100;
	
	{attribute 'TcLinkTo' := '		.arrRaw[0]	:= TIIB(8)^Module 2 (IOL_I_2byte)^TxPDO^input byte 0;	
									.arrRaw[1] 	:= TIIB(8)^Module 2 (IOL_I_2byte)^TxPDO^input byte 1;
									.nState		:= TIIB(8)^IO-Link DeviceState Inputs^Status of IO-Link Port 2;'}
	fbGripperPos2				: FB_MPS100;
END_VAR

// ---- GVLs/GVL_IO_CNC1.TcGVL
VAR_GLOBAL
//(**************************************************Inputs*********************************************************)	
//	// 1.x
//	{attribute 'TcLinkTo' := 'TIIB(13)^Channel 1^Input'} 
//	i_bCnc1ServoInWorkPos1			AT %I*	:BOOL;		// Satu mozgató 1 mh.
//	{attribute 'TcLinkTo' := 'TIIB(13)^Channel 2^Input'}
//	i_bCnc1ServoInBasePos1			AT %I*	:BOOL;		// Satu mozgató 1 ah.
//	{attribute 'TcLinkTo' := 'TIIB(13)^Channel 3^Input'}
//	i_bCnc1ServoInWorkPos2			AT %I*	:BOOL;		// Satu mozgató 2 mh.
//	{attribute 'TcLinkTo' := 'TIIB(13)^Channel 4^Input'}
//	i_bCnc1ServoInBasePos2			AT %I*	:BOOL;		// Satu mozgató 2 ah.
//	{attribute 'TcLinkTo' := 'TIIB(13)^Channel 5^Input'}
//	i_bCnc1ServoLockInWorkPos		AT %I*	:BOOL;		// Satu rögzítő mh.
//	{attribute 'TcLinkTo' := 'TIIB(13)^Channel 6^Input'}
//	i_bCnc1ServoLockInBasePos		AT %I*	:BOOL;		// Satu rögzítő ah.
//	{attribute 'TcLinkTo' := 'TIIB(13)^Channel 7^Input'}
//	i_bCnc1ViseLockInPos			AT %I*	:BOOL;		// Satu rögzítő pozícióban.
//	{attribute 'TcLinkTo' := 'TIIB(13)^Channel 8^Input'}
//	i_bCnc1ToolCheck				AT %I*	:BOOL;		// Szerszámellenörző
	

//(**************************************************Outputs*********************************************************)
//	{attribute 'TcLinkTo' := 'TIIB(14)^Channel 1^Output'}
//	q_bCnc1ServoMoveToWork1			AT %Q*	:BOOL;		// Satu mozgató 1 mh.
//	{attribute 'TcLinkTo' := 'TIIB(14)^Channel 2^Output'}
//	q_bCnc1ServoMoveToBase1			AT %Q*	:BOOL;		// Satu mozgató 1 ah.
//	{attribute 'TcLinkTo' := 'TIIB(14)^Channel 3^Output'}
//	q_bCnc1ServoMoveToWork2			AT %Q*	:BOOL;		// Satu mozgató 2 mh.
//	{attribute 'TcLinkTo' := 'TIIB(14)^Channel 4^Output'}
//	q_bCnc1ServoMoveToBase2			AT %Q*	:BOOL;		// Satu mozgató 2 ah.
//	{attribute 'TcLinkTo' := 'TIIB(14)^Channel 5^Output'}
//	q_bCnc1ServoLiickMoveToWork		AT %Q*	:BOOL;		// Satu rözítő mh. (kioldás)
//	{attribute 'TcLinkTo' := 'TIIB(14)^Channel 6^Output'}
//	q_bCnc1ToolCheckBlower 			AT %Q*	:BOOL;		// Szerszám ellenőrző tisztítás

END_VAR

// ---- GVLs/GVL_Main.TcGVL
VAR_GLOBAL
	// Blink
	bBL50p50						:BOOL; // 50ms/50ms
	bBL100p100						:BOOL; // 100ms/100ms
	bBL250p250						:BOOL; // 250ms/250ms
	bBL500p500						:BOOL; // 500ms/500ms
	bBL1000p1000					:BOOL; // 1000ms/1000ms
	bBL2000p2000					:BOOL; // 2000ms/2000ms
	bBL250p750						:BOOL; // 750ms/250ms
	bBL750p250						:BOOL;
	bTakt100ms						:BOOL; // Takt 100ms
	bTakt200ms						:BOOL; // Takt 200ms
	bTakt500ms						:BOOL; // Takt 500ms
	bTakt1s							:BOOL; // Takt 1000ms

	bFirstCycle						:BOOL := TRUE; 
	wLifeSignal						:WORD;
	bManualModeVise					:BOOL;				(* Manual mode *)
	bManualModeRequestVise			:BOOL;
	sModeVise						:STRING;			(* Actual mode *)
	nModeVise						:BYTE;
	bManualMode						:BOOL;				(* Manual mode *)
	bManualModeRequest				:BOOL;
	sMode							:STRING;			(* Actual mode *)
	nMode							:BYTE;
	bStepMode						:BOOL;				(* Step mode *)
	bStepP							:BOOL;				(* Step pulse *)
	bStepHMI						:BOOL;				(* Step button HMI *)
	bStepEnable						:BOOL;				(* Step enable *)
	bAckHMI							:BOOL;				(* Error acknowledge HMI *)
	bAckP							:BOOL;				(* Acknowledge pulse *)
	bGlobalEHAVise					:BOOL;				(* Error-handling active *)
	bGlobalEHA						:BOOL;				(* Error-handling active *)
	bGlobalError					:BOOL;				(* Global error bit *)
	bDoorOpenReq					:BOOL;				(* Door open request *)
	bInitTCPIP						:BOOL := TRUE;	
	bDrOpenHMI						:BOOL;
	wError							:WORD;
	fbTime 							:FB_LocalSystemTime;
	dtSystemTime					:DATE_AND_TIME;
	fbDoor							:FB_Door;
	aViseStatus						:ARRAY[1..14] OF ST_Vise_Status;
	aViseOrder						:ARRAY[1..14] OF ST_Order;
	
	bStepModeViseStation						:BOOL;				(* Step mode *)
	bStepPViseStation							:BOOL;				(* Step pulse *)
	bStepHMIViseStation						:BOOL;				(* Step button HMI *)
	bStepEnableViseStation						:BOOL;				(* Step enable *)
	
	{attribute 'TcLinkTo' := '		.q_bGreenColor	 := TIIB(85)^IO-Link Port1^Segment 1 -off/on/flash;	
									.q_bYellowColor  := TIIB(85)^IO-Link Port1^Segment 2 -off/on/flash;
									.q_bRedColor	 := TIIB(85)^IO-Link Port1^Segment 3 -off/on/flash;
									.q_bBuzzer		 := TIIB(85)^IO-Link Port1^Segment 4 -off/on/flash;'}
	fbNotSmartLight					:FB_Not_SmartLight;
	
	
	{attribute 'TcLinkTo' := '  [1].fbVise.q_bWorkPos  			:= TIIB(88)^Output1^Outputs^Output 0;
								[1].fbVise.q_bBasePos  			:= TIIB(88)^Output1^Outputs^Output 1;
								[2].fbVise.q_bWorkPos  			:= TIIB(88)^Output1^Outputs^Output 2;
								[2].fbVise.q_bBasePos  			:= TIIB(88)^Output1^Outputs^Output 3;
								[3].fbVise.q_bWorkPos  			:= TIIB(88)^Output1^Outputs^Output 4;
								[3].fbVise.q_bBasePos  			:= TIIB(88)^Output1^Outputs^Output 5;
								[4].fbVise.q_bWorkPos  			:= TIIB(88)^Output1^Outputs^Output 6;
								[4].fbVise.q_bBasePos  			:= TIIB(88)^Output1^Outputs^Output 7;
								[5].fbVise.q_bWorkPos  			:= TIIB(88)^Output2^Outputs^Output 0;
								[5].fbVise.q_bBasePos  			:= TIIB(88)^Output2^Outputs^Output 1;
								[6].fbVise.q_bWorkPos  			:= TIIB(88)^Output2^Outputs^Output 2;
								[6].fbVise.q_bBasePos 			:= TIIB(88)^Output2^Outputs^Output 3;
								[7].fbVise.q_bWorkPos 			:= TIIB(88)^Output2^Outputs^Output 4;
								[7].fbVise.q_bBasePos 			:= TIIB(88)^Output2^Outputs^Output 5;
								[1].fbStopper_In.q_bWorkPos		:= TIIB(88)^Output3^Outputs^Output 0;
								[1].fbStopper_Out.q_bWorkPos  	:= TIIB(88)^Output3^Outputs^Output 2;
								[2].fbStopper_In.q_bWorkPos 	:= TIIB(88)^Output3^Outputs^Output 4;
								[2].fbStopper_Out.q_bWorkPos 	:= TIIB(88)^Output3^Outputs^Output 6;
								[3].fbStopper_In.q_bWorkPos  	:= TIIB(88)^Output4^Outputs^Output 0;
								[3].fbStopper_Out.q_bWorkPos  	:= TIIB(88)^Output4^Outputs^Output 2;
								[4].fbStopper_In.q_bWorkPos  	:= TIIB(88)^Output4^Outputs^Output 4;
								[4].fbStopper_Out.q_bWorkPos  	:= TIIB(88)^Output4^Outputs^Output 6;
								[5].fbStopper_In.q_bWorkPos  	:= TIIB(88)^Output5^Outputs^Output 0;
								[5].fbStopper_Out.q_bWorkPos  	:= TIIB(88)^Output5^Outputs^Output 2;
								[6].fbStopper_In.q_bWorkPos  	:= TIIB(88)^Output5^Outputs^Output 4;
								[6].fbStopper_Out.q_bWorkPos  	:= TIIB(88)^Output5^Outputs^Output 6;
								[7].fbStopper_In.q_bWorkPos  	:= TIIB(88)^Output6^Outputs^Output 0;
								[7].fbStopper_Out.q_bWorkPos  	:= TIIB(88)^Output6^Outputs^Output 2;
								[8].fbVise.q_bWorkPos  			:= TIIB(89)^Output1^Outputs^Output 0;
								[8].fbVise.q_bBasePos  			:= TIIB(89)^Output1^Outputs^Output 1;
								[9].fbVise.q_bWorkPos  			:= TIIB(89)^Output1^Outputs^Output 2;
								[9].fbVise.q_bBasePos  			:= TIIB(89)^Output1^Outputs^Output 3;
								[10].fbVise.q_bWorkPos  		:= TIIB(89)^Output1^Outputs^Output 4;
								[10].fbVise.q_bBasePos  		:= TIIB(89)^Output1^Outputs^Output 5;
								[11].fbVise.q_bWorkPos  		:= TIIB(89)^Output1^Outputs^Output 6;
								[11].fbVise.q_bBasePos  		:= TIIB(89)^Output1^Outputs^Output 7;
								[12].fbVise.q_bWorkPos  		:= TIIB(89)^Output2^Outputs^Output 0;
								[12].fbVise.q_bBasePos  		:= TIIB(89)^Output2^Outputs^Output 1;
								[13].fbVise.q_bWorkPos  		:= TIIB(89)^Output2^Outputs^Output 2;
								[13].fbVise.q_bBasePos 			:= TIIB(89)^Output2^Outputs^Output 3;
								[14].fbVise.q_bWorkPos 			:= TIIB(89)^Output2^Outputs^Output 4;
								[14].fbVise.q_bBasePos 			:= TIIB(89)^Output2^Outputs^Output 5;
								[8].fbStopper_In.q_bWorkPos		:= TIIB(89)^Output3^Outputs^Output 0;
								[8].fbStopper_Out.q_bWorkPos  	:= TIIB(89)^Output3^Outputs^Output 2;
								[9].fbStopper_In.q_bWorkPos 	:= TIIB(89)^Output3^Outputs^Output 4;
								[9].fbStopper_Out.q_bWorkPos 	:= TIIB(89)^Output3^Outputs^Output 6;
								[10].fbStopper_In.q_bWorkPos  	:= TIIB(89)^Output4^Outputs^Output 0;
								[10].fbStopper_Out.q_bWorkPos  	:= TIIB(89)^Output4^Outputs^Output 2;
								[11].fbStopper_In.q_bWorkPos  	:= TIIB(89)^Output4^Outputs^Output 4;
								[11].fbStopper_Out.q_bWorkPos  	:= TIIB(89)^Output4^Outputs^Output 6;
								[12].fbStopper_In.q_bWorkPos  	:= TIIB(89)^Output5^Outputs^Output 0;
								[12].fbStopper_Out.q_bWorkPos  	:= TIIB(89)^Output5^Outputs^Output 2;
								[13].fbStopper_In.q_bWorkPos  	:= TIIB(89)^Output5^Outputs^Output 4;
								[13].fbStopper_Out.q_bWorkPos  	:= TIIB(89)^Output5^Outputs^Output 6;
								[14].fbStopper_In.q_bWorkPos  	:= TIIB(89)^Output6^Outputs^Output 0;
								[14].fbStopper_Out.q_bWorkPos  	:= TIIB(89)^Output6^Outputs^Output 2;'}													
	fbViseStation				:ARRAY[1..14] OF FB_Vise_Station;	
	{attribute 'TcLinkTo' := 'TIIB(71)^Output2^Outputs^Output 6'}
	q_bViseOut_1_7		AT %Q*	:BOOL;	
	{attribute 'TcLinkTo' := 'TIIB(72)^Output2^Outputs^Output 6'}
	q_bViseOut_8_14		AT %Q*	:BOOL;	
	
	
	// RGB
	{attribute 'TcLinkTo' := '	.i_stRGB_In.LifeSig := TIIB(87)^Inputs^LifeSignal;
								.i_stRGB_In.Resp := TIIB(87)^Inputs^Response;
								.q_stRGB_Out.LifeSig := TIIB(87)^Outputs^LifeSignal;
								.q_stRGB_Out.Command := TIIB(87)^Outputs^Command;
								.q_stRGB_Out.arrRGB[1] := TIIB(87)^Outputs^RGB_01;
								.q_stRGB_Out.arrRGB[2] := TIIB(87)^Outputs^RGB_02;
								.q_stRGB_Out.arrRGB[3] := TIIB(87)^Outputs^RGB_03;
								.q_stRGB_Out.arrRGB[4] := TIIB(87)^Outputs^RGB_04;
								.q_stRGB_Out.arrRGB[5] := TIIB(87)^Outputs^RGB_05;
								.q_stRGB_Out.arrRGB[6] := TIIB(87)^Outputs^RGB_06;
								.q_stRGB_Out.arrRGB[7] := TIIB(87)^Outputs^RGB_07;
								.q_stRGB_Out.arrRGB[8] := TIIB(87)^Outputs^RGB_08;
								.q_stRGB_Out.arrRGB[9] := TIIB(87)^Outputs^RGB_09;
								.q_stRGB_Out.arrRGB[10] := TIIB(87)^Outputs^RGB_10;
								.q_stRGB_Out.arrRGB[11] := TIIB(87)^Outputs^RGB_11;
								.q_stRGB_Out.arrRGB[12] := TIIB(87)^Outputs^RGB_12;
								.q_stRGB_Out.arrRGB[13] := TIIB(87)^Outputs^RGB_13;
								.q_stRGB_Out.arrRGB[14] := TIIB(87)^Outputs^RGB_14;
								.q_stRGB_Out.arrRGB[15] := TIIB(87)^Outputs^RGB_15;
								.q_stRGB_Out.arrRGB[16] := TIIB(87)^Outputs^RGB_16;
								.q_stRGB_Out.arrRGB[17] := TIIB(87)^Outputs^RGB_17;
								.q_stRGB_Out.arrRGB[18] := TIIB(87)^Outputs^RGB_18;
								.q_stRGB_Out.arrRGB[19] := TIIB(87)^Outputs^RGB_19;
								.q_stRGB_Out.arrRGB[20] := TIIB(87)^Outputs^RGB_20;
								.q_stRGB_Out.arrRGB[21] := TIIB(87)^Outputs^RGB_21;
								.q_stRGB_Out.arrRGB[22] := TIIB(87)^Outputs^RGB_22;
								.q_stRGB_Out.arrRGB[23] := TIIB(87)^Outputs^RGB_23;
								.q_stRGB_Out.arrRGB[24] := TIIB(87)^Outputs^RGB_24;'}
	fbRgbLights					:FB_RGB_Light;

	fb3DCam					:FB_TCP_IP_Comm;
END_VAR

// ---- GVLs/GVL_Palette.TcGVL
VAR_GLOBAL PERSISTENT
	arrPalette					: ARRAY [0..200] OF ST_Dut_Data;
END_VAR

// ---- GVLs/GVL_Python.TcGVL
{attribute 'qualified_only'}
VAR_GLOBAL
	nLifeSignal				: WORD;
END_VAR

